(* Check controller alarm *)
IF sREL_ALM<>REL_ALM THEN
	CASE REL_ALM OF
		0: IF NOT chkREL_ST.OUT THEN LogEv(EL_Log,EO_LUXM,ID,1,''); END_IF
		1: LogEv(EL_Alarm,EO_LUXM,ID,6,'');
		2: LogEv(EL_Wrn  ,EO_LUXM,ID,4,WORD_TO_STRING(REL_A));
		3: LogEv(EL_Wrn  ,EO_LUXM,ID,5,WORD_TO_STRING(REL_A));
		4: LogEv(EL_Alarm,EO_LUXM,ID,7,WORD_TO_STRING(REL_A));
		5: LogEv(EL_Alarm,EO_LUXM,ID,8,'');
	END_CASE
	sREL_ALM:=REL_ALM;
END_IF

(* Status color *)
   IF REL_ALM=1 OR REL_ALM>3 OR chkREL_ST.OUT	THEN Status_Log:=2; Status_Vis:=COLOR_RED;
ELSIF REL_ALM<>0								THEN Status_Log:=1; Status_Vis:=COLOR_YELLOW;
                  	   							ELSE Status_Log:=0; Status_Vis:=SEL(REL_EN,COLOR_GREEN_OFF,COLOR_GREEN);
END_IF

ACTION AddLogData:
Logger.s1:=INSERT('&LUXM=',BYTE_TO_STRING(ID),5);
IF ID<10 THEN Logger.s1:=INSERT(Logger.s1,'0',5); END_IF

Logger.s1:=CONCAT(Logger.s1,WORD_TO_STRING(REL_V));				Logger.s1:=CONCAT(Logger.s1,';');
Logger.s1:=CONCAT(Logger.s1,WORD_TO_STRING(REL_A));				Logger.s1:=CONCAT(Logger.s1,';');
Logger.s1:=CONCAT(Logger.s1,DWORD_TO_STRING(ENERGYCOUNTER));	Logger.s1:=CONCAT(Logger.s1,';');
Logger.s1:=CONCAT(Logger.s1,DWORD_TO_STRING(WORKINGTIME));		Logger.s1:=CONCAT(Logger.s1,';');
Logger.s1:=CONCAT(Logger.s1,DWORD_TO_STRING(POWERONCYCLES));	Logger.s1:=CONCAT(Logger.s1,';');
Logger.s1:=CONCAT(Logger.s1,INT_TO_STRING(REL_TEMP));			Logger.s1:=CONCAT(Logger.s1,';');

Logger.s1:=CONCAT(Logger.s1,BYTE_TO_STRING(Status_Log));
ADDSTRING(ADR(Logger.TData), ADR(Logger.s1), Logger.TLen);
END_ACTION

ACTION StatReset:
(* Reset statistic counters *)
WORKINGTIME:=0;
POWERONCYCLES:=0;
ENERGYCOUNTER:=0;
END_ACTION

END_FUNCTION_BLOCK

// AC14nn/Application/VIS_CHONOEDITOR
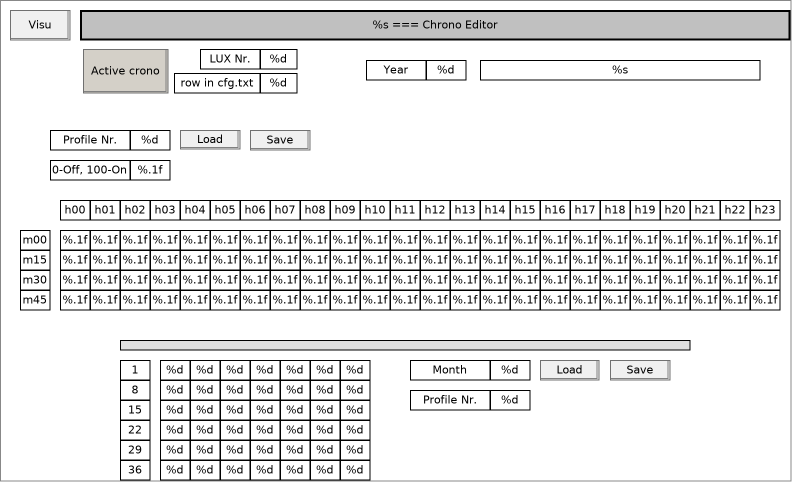
VISUALIZATION VIS_CHONOEDITOR  // 792x482
VAR_IN_OUT
//	x	: word;
//	LuxSel	: word;	
END_VAR
    Rectangle (200,49 60x20), "LUX Nr."
    Rectangle (260,49 37x20), "%d", text variable: CronEd.CN_Sel, colour toggle: CronEd.CN_Sel<>CronEd.CN_Act
        OnMouseDown: write the text variable via Edit, min 1, max 900, title '1'
    Rectangle (50,130 80x20), "Profile Nr."
    Rectangle (130,130 40x20), "%d", text variable: CronEd.PR_Sel, colour toggle: CronEd.PR_Sel<>CronEd.PR_Act
        OnMouseDown: write the text variable via Edit, min 1, max 10
    Rectangle (50,160 80x20), "0-Off, 100-On"
    Rectangle (130,160 40x20), "%.1f", text variable: CronEd.PR_TT
        OnMouseDown: write the text variable via Edit
    Button (180,130 60x19), "Load", pressed state: CronEd.PR_Load
        toggle CronEd.PR_Load
    Button (250,130 60x20), "Save", pressed state: CronEd.PR_Save
        toggle CronEd.PR_Save
    Rectangle (20,230 30x20), "m00"
    Rectangle (20,250 30x20), "m15"
    Rectangle (20,270 30x20), "m30"
    Rectangle (20,290 30x20), "m45"
    Rectangle (80,10 710x30), "%s === Chrono Editor", text variable: Plant_NAME
    Button (10,10 60x30), "Visu"
        OnMouseUp:  Assign=PLC_Visualization, Type=Assignment
    Polygon (20,210)
    RoundedRectangle (60,230 30x20), "%.1f", text variable: INT_TO_REAL(CronEd.PR.Setpoint[0])/10
        OnMouseUp: execute { CronEd.PR.Setpoint[0]:=(REAL_TO_WORD(CronEd.PR_TT*10)); }
    RoundedRectangle (60,250 30x20), "%.1f", text variable: INT_TO_REAL(CronEd.PR.Setpoint[1])/10
        OnMouseUp: execute { CronEd.PR.Setpoint[1]:=(REAL_TO_WORD(CronEd.PR_TT*10)); }
    RoundedRectangle (60,270 30x20), "%.1f", text variable: INT_TO_REAL(CronEd.PR.Setpoint[2])/10
        OnMouseUp: execute { CronEd.PR.Setpoint[2]:=(REAL_TO_WORD(CronEd.PR_TT*10)); }
    RoundedRectangle (60,290 30x20), "%.1f", text variable: INT_TO_REAL(CronEd.PR.Setpoint[3])/10
        OnMouseUp: execute { CronEd.PR.Setpoint[3]:=(REAL_TO_WORD(CronEd.PR_TT*10)); }
    Rectangle (60,200 30x20), "h00"
        OnMouseUp: execute { CronEd.PR.Setpoint[0]:=(REAL_TO_WORD(CronEd.PR_TT*10)); }
        OnMouseUp: execute { CronEd.PR.Setpoint[1]:=(REAL_TO_WORD(CronEd.PR_TT*10)); }
        OnMouseUp: execute { CronEd.PR.Setpoint[2]:=(REAL_TO_WORD(CronEd.PR_TT*10)); }
        OnMouseUp: execute { CronEd.PR.Setpoint[3]:=(REAL_TO_WORD(CronEd.PR_TT*10)); }
    RoundedRectangle (90,230 30x20), "%.1f", text variable: INT_TO_REAL(CronEd.PR.Setpoint[4])/10
        OnMouseUp: execute { CronEd.PR.Setpoint[4]:=(REAL_TO_WORD(CronEd.PR_TT*10)); }
    RoundedRectangle (90,250 30x20), "%.1f", text variable: INT_TO_REAL(CronEd.PR.Setpoint[5])/10
        OnMouseUp: execute { CronEd.PR.Setpoint[5]:=(REAL_TO_WORD(CronEd.PR_TT*10)); }
    RoundedRectangle (90,270 30x20), "%.1f", text variable: INT_TO_REAL(CronEd.PR.Setpoint[6])/10
        OnMouseUp: execute { CronEd.PR.Setpoint[6]:=(REAL_TO_WORD(CronEd.PR_TT*10)); }
    RoundedRectangle (90,290 30x20), "%.1f", text variable: INT_TO_REAL(CronEd.PR.Setpoint[7])/10
        OnMouseUp: execute { CronEd.PR.Setpoint[7]:=(REAL_TO_WORD(CronEd.PR_TT*10)); }
    Rectangle (90,200 30x20), "h01"
        OnMouseUp: execute { CronEd.PR.Setpoint[4]:=(REAL_TO_WORD(CronEd.PR_TT*10)); }
        OnMouseUp: execute { CronEd.PR.Setpoint[5]:=(REAL_TO_WORD(CronEd.PR_TT*10)); }
        OnMouseUp: execute { CronEd.PR.Setpoint[6]:=(REAL_TO_WORD(CronEd.PR_TT*10)); }
        OnMouseUp: execute { CronEd.PR.Setpoint[7]:=(REAL_TO_WORD(CronEd.PR_TT*10)); }
    RoundedRectangle (120,230 30x20), "%.1f", text variable: INT_TO_REAL(CronEd.PR.Setpoint[8])/10
        OnMouseUp: execute { CronEd.PR.Setpoint[8]:=(REAL_TO_WORD(CronEd.PR_TT*10)); }
    RoundedRectangle (120,250 30x20), "%.1f", text variable: INT_TO_REAL(CronEd.PR.Setpoint[9])/10
        OnMouseUp: execute { CronEd.PR.Setpoint[9]:=(REAL_TO_WORD(CronEd.PR_TT*10)); }
    RoundedRectangle (120,270 30x20), "%.1f", text variable: INT_TO_REAL(CronEd.PR.Setpoint[10])/10
        OnMouseUp: execute { CronEd.PR.Setpoint[10]:=(REAL_TO_WORD(CronEd.PR_TT*10)); }
    RoundedRectangle (120,290 30x20), "%.1f", text variable: INT_TO_REAL(CronEd.PR.Setpoint[11])/10
        OnMouseUp: execute { CronEd.PR.Setpoint[11]:=(REAL_TO_WORD(CronEd.PR_TT*10)); }
    Rectangle (120,200 30x20), "h02"
        OnMouseUp: execute { CronEd.PR.Setpoint[8]:=(REAL_TO_WORD(CronEd.PR_TT*10)); }
        OnMouseUp: execute { CronEd.PR.Setpoint[9]:=(REAL_TO_WORD(CronEd.PR_TT*10)); }
        OnMouseUp: execute { CronEd.PR.Setpoint[10]:=(REAL_TO_WORD(CronEd.PR_TT*10)); }
        OnMouseUp: execute { CronEd.PR.Setpoint[11]:=(REAL_TO_WORD(CronEd.PR_TT*10)); }
    RoundedRectangle (150,230 30x20), "%.1f", text variable: INT_TO_REAL(CronEd.PR.Setpoint[12])/10
        OnMouseUp: execute { CronEd.PR.Setpoint[12]:=(REAL_TO_WORD(CronEd.PR_TT*10)); }
    RoundedRectangle (150,250 30x20), "%.1f", text variable: INT_TO_REAL(CronEd.PR.Setpoint[13])/10
        OnMouseUp: execute { CronEd.PR.Setpoint[13]:=(REAL_TO_WORD(CronEd.PR_TT*10)); }
    RoundedRectangle (150,270 30x20), "%.1f", text variable: INT_TO_REAL(CronEd.PR.Setpoint[14])/10
        OnMouseUp: execute { CronEd.PR.Setpoint[14]:=(REAL_TO_WORD(CronEd.PR_TT*10)); }
    RoundedRectangle (150,290 30x20), "%.1f", text variable: INT_TO_REAL(CronEd.PR.Setpoint[15])/10
        OnMouseUp: execute { CronEd.PR.Setpoint[15]:=(REAL_TO_WORD(CronEd.PR_TT*10)); }
    Rectangle (150,200 30x20), "h03"
        OnMouseUp: execute { CronEd.PR.Setpoint[15]:=(REAL_TO_WORD(CronEd.PR_TT*10)); }
        OnMouseUp: execute { CronEd.PR.Setpoint[14]:=(REAL_TO_WORD(CronEd.PR_TT*10)); }
        OnMouseUp: execute { CronEd.PR.Setpoint[13]:=(REAL_TO_WORD(CronEd.PR_TT*10)); }
        OnMouseUp: execute { CronEd.PR.Setpoint[12]:=(REAL_TO_WORD(CronEd.PR_TT*10)); }
    RoundedRectangle (180,230 30x20), "%.1f", text variable: INT_TO_REAL(CronEd.PR.Setpoint[16])/10
        OnMouseUp: execute { CronEd.PR.Setpoint[16]:=(REAL_TO_WORD(CronEd.PR_TT*10)); }
    RoundedRectangle (180,250 30x20), "%.1f", text variable: INT_TO_REAL(CronEd.PR.Setpoint[17])/10
        OnMouseUp: execute { CronEd.PR.Setpoint[17]:=(REAL_TO_WORD(CronEd.PR_TT*10)); }
    RoundedRectangle (180,270 30x20), "%.1f", text variable: INT_TO_REAL(CronEd.PR.Setpoint[18])/10
        OnMouseUp: execute { CronEd.PR.Setpoint[18]:=(REAL_TO_WORD(CronEd.PR_TT*10)); }
    RoundedRectangle (180,290 30x20), "%.1f", text variable: INT_TO_REAL(CronEd.PR.Setpoint[19])/10
        OnMouseUp: execute { CronEd.PR.Setpoint[19]:=(REAL_TO_WORD(CronEd.PR_TT*10)); }
    Rectangle (180,200 30x20), "h04"
        OnMouseUp: execute { CronEd.PR.Setpoint[19]:=(REAL_TO_WORD(CronEd.PR_TT*10)); }
        OnMouseUp: execute { CronEd.PR.Setpoint[18]:=(REAL_TO_WORD(CronEd.PR_TT*10)); }
        OnMouseUp: execute { CronEd.PR.Setpoint[17]:=(REAL_TO_WORD(CronEd.PR_TT*10)); }
        OnMouseUp: execute { CronEd.PR.Setpoint[16]:=(REAL_TO_WORD(CronEd.PR_TT*10)); }
    RoundedRectangle (210,230 30x20), "%.1f", text variable: INT_TO_REAL(CronEd.PR.Setpoint[20])/10
        OnMouseUp: execute { CronEd.PR.Setpoint[20]:=(REAL_TO_WORD(CronEd.PR_TT*10)); }
    RoundedRectangle (210,250 30x20), "%.1f", text variable: INT_TO_REAL(CronEd.PR.Setpoint[21])/10
        OnMouseUp: execute { CronEd.PR.Setpoint[21]:=(REAL_TO_WORD(CronEd.PR_TT*10)); }
    RoundedRectangle (210,270 30x20), "%.1f", text variable: INT_TO_REAL(CronEd.PR.Setpoint[22])/10
        OnMouseUp: execute { CronEd.PR.Setpoint[22]:=(REAL_TO_WORD(CronEd.PR_TT*10)); }
    RoundedRectangle (210,290 30x20), "%.1f", text variable: INT_TO_REAL(CronEd.PR.Setpoint[23])/10
        OnMouseUp: execute { CronEd.PR.Setpoint[23]:=(REAL_TO_WORD(CronEd.PR_TT*10)); }
    Rectangle (210,200 30x20), "h05"
        OnMouseUp: execute { CronEd.PR.Setpoint[23]:=(REAL_TO_WORD(CronEd.PR_TT*10)); }
        OnMouseUp: execute { CronEd.PR.Setpoint[22]:=(REAL_TO_WORD(CronEd.PR_TT*10)); }
        OnMouseUp: execute { CronEd.PR.Setpoint[21]:=(REAL_TO_WORD(CronEd.PR_TT*10)); }
        OnMouseUp: execute { CronEd.PR.Setpoint[20]:=(REAL_TO_WORD(CronEd.PR_TT*10)); }
    RoundedRectangle (240,230 30x20), "%.1f", text variable: INT_TO_REAL(CronEd.PR.Setpoint[24])/10
        OnMouseUp: execute { CronEd.PR.Setpoint[24]:=(REAL_TO_WORD(CronEd.PR_TT*10)); }
    RoundedRectangle (240,250 30x20), "%.1f", text variable: INT_TO_REAL(CronEd.PR.Setpoint[25])/10
        OnMouseUp: execute { CronEd.PR.Setpoint[25]:=(REAL_TO_WORD(CronEd.PR_TT*10)); }
    RoundedRectangle (240,270 30x20), "%.1f", text variable: INT_TO_REAL(CronEd.PR.Setpoint[26])/10
        OnMouseUp: execute { CronEd.PR.Setpoint[26]:=(REAL_TO_WORD(CronEd.PR_TT*10)); }
    RoundedRectangle (240,290 30x20), "%.1f", text variable: INT_TO_REAL(CronEd.PR.Setpoint[27])/10
        OnMouseUp: execute { CronEd.PR.Setpoint[27]:=(REAL_TO_WORD(CronEd.PR_TT*10)); }
    Rectangle (240,200 30x20), "h06"
        OnMouseUp: execute { CronEd.PR.Setpoint[27]:=(REAL_TO_WORD(CronEd.PR_TT*10)); }
        OnMouseUp: execute { CronEd.PR.Setpoint[26]:=(REAL_TO_WORD(CronEd.PR_TT*10)); }
        OnMouseUp: execute { CronEd.PR.Setpoint[25]:=(REAL_TO_WORD(CronEd.PR_TT*10)); }
        OnMouseUp: execute { CronEd.PR.Setpoint[24]:=(REAL_TO_WORD(CronEd.PR_TT*10)); }
    RoundedRectangle (270,230 30x20), "%.1f", text variable: INT_TO_REAL(CronEd.PR.Setpoint[28])/10
        OnMouseUp: execute { CronEd.PR.Setpoint[28]:=(REAL_TO_WORD(CronEd.PR_TT*10)); }
    RoundedRectangle (270,250 30x20), "%.1f", text variable: INT_TO_REAL(CronEd.PR.Setpoint[29])/10
        OnMouseUp: execute { CronEd.PR.Setpoint[29]:=(REAL_TO_WORD(CronEd.PR_TT*10)); }
    RoundedRectangle (270,270 30x20), "%.1f", text variable: INT_TO_REAL(CronEd.PR.Setpoint[30])/10
        OnMouseUp: execute { CronEd.PR.Setpoint[30]:=(REAL_TO_WORD(CronEd.PR_TT*10)); }
    RoundedRectangle (270,290 30x20), "%.1f", text variable: INT_TO_REAL(CronEd.PR.Setpoint[31])/10
        OnMouseUp: execute { CronEd.PR.Setpoint[31]:=(REAL_TO_WORD(CronEd.PR_TT*10)); }
    Rectangle (270,200 30x20), "h07"
        OnMouseUp: execute { CronEd.PR.Setpoint[31]:=(REAL_TO_WORD(CronEd.PR_TT*10)); }
        OnMouseUp: execute { CronEd.PR.Setpoint[30]:=(REAL_TO_WORD(CronEd.PR_TT*10)); }
        OnMouseUp: execute { CronEd.PR.Setpoint[29]:=(REAL_TO_WORD(CronEd.PR_TT*10)); }
        OnMouseUp: execute { CronEd.PR.Setpoint[28]:=(REAL_TO_WORD(CronEd.PR_TT*10)); }
    RoundedRectangle (300,230 30x20), "%.1f", text variable: INT_TO_REAL(CronEd.PR.Setpoint[32])/10
        OnMouseUp: execute { CronEd.PR.Setpoint[32]:=(REAL_TO_WORD(CronEd.PR_TT*10)); }
    RoundedRectangle (300,250 30x20), "%.1f", text variable: INT_TO_REAL(CronEd.PR.Setpoint[33])/10
        OnMouseUp: execute { CronEd.PR.Setpoint[33]:=(REAL_TO_WORD(CronEd.PR_TT*10)); }
    RoundedRectangle (300,270 30x20), "%.1f", text variable: INT_TO_REAL(CronEd.PR.Setpoint[34])/10
        OnMouseUp: execute { CronEd.PR.Setpoint[34]:=(REAL_TO_WORD(CronEd.PR_TT*10)); }
    RoundedRectangle (300,290 30x20), "%.1f", text variable: INT_TO_REAL(CronEd.PR.Setpoint[35])/10
        OnMouseUp: execute { CronEd.PR.Setpoint[35]:=(REAL_TO_WORD(CronEd.PR_TT*10)); }
    Rectangle (300,200 30x20), "h08"
        OnMouseUp: execute { CronEd.PR.Setpoint[35]:=(REAL_TO_WORD(CronEd.PR_TT*10)); }
        OnMouseUp: execute { CronEd.PR.Setpoint[34]:=(REAL_TO_WORD(CronEd.PR_TT*10)); }
        OnMouseUp: execute { CronEd.PR.Setpoint[33]:=(REAL_TO_WORD(CronEd.PR_TT*10)); }
        OnMouseUp: execute { CronEd.PR.Setpoint[32]:=(REAL_TO_WORD(CronEd.PR_TT*10)); }
    RoundedRectangle (330,230 30x20), "%.1f", text variable: INT_TO_REAL(CronEd.PR.Setpoint[36])/10
        OnMouseUp: execute { CronEd.PR.Setpoint[36]:=(REAL_TO_WORD(CronEd.PR_TT*10)); }
    RoundedRectangle (330,250 30x20), "%.1f", text variable: INT_TO_REAL(CronEd.PR.Setpoint[37])/10
        OnMouseUp: execute { CronEd.PR.Setpoint[37]:=(REAL_TO_WORD(CronEd.PR_TT*10)); }
    RoundedRectangle (330,270 30x20), "%.1f", text variable: INT_TO_REAL(CronEd.PR.Setpoint[38])/10
        OnMouseUp: execute { CronEd.PR.Setpoint[38]:=(REAL_TO_WORD(CronEd.PR_TT*10)); }
    RoundedRectangle (330,290 30x20), "%.1f", text variable: INT_TO_REAL(CronEd.PR.Setpoint[39])/10
        OnMouseUp: execute { CronEd.PR.Setpoint[39]:=(REAL_TO_WORD(CronEd.PR_TT*10)); }
    Rectangle (330,200 30x20), "h09"
        OnMouseUp: execute { CronEd.PR.Setpoint[39]:=(REAL_TO_WORD(CronEd.PR_TT*10)); }
        OnMouseUp: execute { CronEd.PR.Setpoint[38]:=(REAL_TO_WORD(CronEd.PR_TT*10)); }
        OnMouseUp: execute { CronEd.PR.Setpoint[37]:=(REAL_TO_WORD(CronEd.PR_TT*10)); }
        OnMouseUp: execute { CronEd.PR.Setpoint[36]:=(REAL_TO_WORD(CronEd.PR_TT*10)); }
    RoundedRectangle (360,230 30x20), "%.1f", text variable: INT_TO_REAL(CronEd.PR.Setpoint[40])/10
        OnMouseUp: execute { CronEd.PR.Setpoint[40]:=(REAL_TO_WORD(CronEd.PR_TT*10)); }
    RoundedRectangle (360,250 30x20), "%.1f", text variable: INT_TO_REAL(CronEd.PR.Setpoint[41])/10
        OnMouseUp: execute { CronEd.PR.Setpoint[41]:=(REAL_TO_WORD(CronEd.PR_TT*10)); }
    RoundedRectangle (360,270 30x20), "%.1f", text variable: INT_TO_REAL(CronEd.PR.Setpoint[42])/10
        OnMouseUp: execute { CronEd.PR.Setpoint[42]:=(REAL_TO_WORD(CronEd.PR_TT*10)); }
    RoundedRectangle (360,290 30x20), "%.1f", text variable: INT_TO_REAL(CronEd.PR.Setpoint[43])/10
        OnMouseUp: execute { CronEd.PR.Setpoint[43]:=(REAL_TO_WORD(CronEd.PR_TT*10)); }
    Rectangle (360,200 30x20), "h10"
        OnMouseUp: execute { CronEd.PR.Setpoint[43]:=(REAL_TO_WORD(CronEd.PR_TT*10)); }
        OnMouseUp: execute { CronEd.PR.Setpoint[42]:=(REAL_TO_WORD(CronEd.PR_TT*10)); }
        OnMouseUp: execute { CronEd.PR.Setpoint[41]:=(REAL_TO_WORD(CronEd.PR_TT*10)); }
        OnMouseUp: execute { CronEd.PR.Setpoint[40]:=(REAL_TO_WORD(CronEd.PR_TT*10)); }
    RoundedRectangle (390,230 30x20), "%.1f", text variable: INT_TO_REAL(CronEd.PR.Setpoint[44])/10
        OnMouseUp: execute { CronEd.PR.Setpoint[44]:=(REAL_TO_WORD(CronEd.PR_TT*10)); }
    RoundedRectangle (390,250 30x20), "%.1f", text variable: INT_TO_REAL(CronEd.PR.Setpoint[45])/10
        OnMouseUp: execute { CronEd.PR.Setpoint[45]:=(REAL_TO_WORD(CronEd.PR_TT*10)); }
    RoundedRectangle (390,270 30x20), "%.1f", text variable: INT_TO_REAL(CronEd.PR.Setpoint[46])/10
        OnMouseUp: execute { CronEd.PR.Setpoint[46]:=(REAL_TO_WORD(CronEd.PR_TT*10)); }
    RoundedRectangle (390,290 30x20), "%.1f", text variable: INT_TO_REAL(CronEd.PR.Setpoint[47])/10
        OnMouseUp: execute { CronEd.PR.Setpoint[47]:=(REAL_TO_WORD(CronEd.PR_TT*10)); }
    Rectangle (390,200 30x20), "h11"
        OnMouseUp: execute { CronEd.PR.Setpoint[47]:=(REAL_TO_WORD(CronEd.PR_TT*10)); }
        OnMouseUp: execute { CronEd.PR.Setpoint[46]:=(REAL_TO_WORD(CronEd.PR_TT*10)); }
        OnMouseUp: execute { CronEd.PR.Setpoint[45]:=(REAL_TO_WORD(CronEd.PR_TT*10)); }
        OnMouseUp: execute { CronEd.PR.Setpoint[44]:=(REAL_TO_WORD(CronEd.PR_TT*10)); }
    RoundedRectangle (420,230 30x20), "%.1f", text variable: INT_TO_REAL(CronEd.PR.Setpoint[48])/10
        OnMouseUp: execute { CronEd.PR.Setpoint[48]:=(REAL_TO_WORD(CronEd.PR_TT*10)); }
    RoundedRectangle (420,250 30x20), "%.1f", text variable: INT_TO_REAL(CronEd.PR.Setpoint[49])/10
        OnMouseUp: execute { CronEd.PR.Setpoint[49]:=(REAL_TO_WORD(CronEd.PR_TT*10)); }
    RoundedRectangle (420,270 30x20), "%.1f", text variable: INT_TO_REAL(CronEd.PR.Setpoint[50])/10
        OnMouseUp: execute { CronEd.PR.Setpoint[50]:=(REAL_TO_WORD(CronEd.PR_TT*10)); }
    RoundedRectangle (420,290 30x20), "%.1f", text variable: INT_TO_REAL(CronEd.PR.Setpoint[51])/10
        OnMouseUp: execute { CronEd.PR.Setpoint[51]:=(REAL_TO_WORD(CronEd.PR_TT*10)); }
    Rectangle (420,200 30x20), "h12"
        OnMouseUp: execute { CronEd.PR.Setpoint[51]:=(REAL_TO_WORD(CronEd.PR_TT*10)); }
        OnMouseUp: execute { CronEd.PR.Setpoint[50]:=(REAL_TO_WORD(CronEd.PR_TT*10)); }
        OnMouseUp: execute { CronEd.PR.Setpoint[49]:=(REAL_TO_WORD(CronEd.PR_TT*10)); }
        OnMouseUp: execute { CronEd.PR.Setpoint[48]:=(REAL_TO_WORD(CronEd.PR_TT*10)); }
    RoundedRectangle (450,230 30x20), "%.1f", text variable: INT_TO_REAL(CronEd.PR.Setpoint[52])/10
        OnMouseUp: execute { CronEd.PR.Setpoint[52]:=(REAL_TO_WORD(CronEd.PR_TT*10)); }
    RoundedRectangle (450,250 30x20), "%.1f", text variable: INT_TO_REAL(CronEd.PR.Setpoint[53])/10
        OnMouseUp: execute { CronEd.PR.Setpoint[53]:=(REAL_TO_WORD(CronEd.PR_TT*10)); }
    RoundedRectangle (450,270 30x20), "%.1f", text variable: INT_TO_REAL(CronEd.PR.Setpoint[54])/10
        OnMouseUp: execute { CronEd.PR.Setpoint[54]:=(REAL_TO_WORD(CronEd.PR_TT*10)); }
    RoundedRectangle (450,290 30x20), "%.1f", text variable: INT_TO_REAL(CronEd.PR.Setpoint[55])/10
        OnMouseUp: execute { CronEd.PR.Setpoint[55]:=(REAL_TO_WORD(CronEd.PR_TT*10)); }
    Rectangle (450,200 30x20), "h13"
        OnMouseUp: execute { CronEd.PR.Setpoint[55]:=(REAL_TO_WORD(CronEd.PR_TT*10)); }
        OnMouseUp: execute { CronEd.PR.Setpoint[54]:=(REAL_TO_WORD(CronEd.PR_TT*10)); }
        OnMouseUp: execute { CronEd.PR.Setpoint[53]:=(REAL_TO_WORD(CronEd.PR_TT*10)); }
        OnMouseUp: execute { CronEd.PR.Setpoint[52]:=(REAL_TO_WORD(CronEd.PR_TT*10)); }
    RoundedRectangle (480,230 30x20), "%.1f", text variable: INT_TO_REAL(CronEd.PR.Setpoint[56])/10
        OnMouseUp: execute { CronEd.PR.Setpoint[56]:=(REAL_TO_WORD(CronEd.PR_TT*10)); }
    RoundedRectangle (480,250 30x20), "%.1f", text variable: INT_TO_REAL(CronEd.PR.Setpoint[57])/10
        OnMouseUp: execute { CronEd.PR.Setpoint[57]:=(REAL_TO_WORD(CronEd.PR_TT*10)); }
    RoundedRectangle (480,270 30x20), "%.1f", text variable: INT_TO_REAL(CronEd.PR.Setpoint[58])/10
        OnMouseUp: execute { CronEd.PR.Setpoint[58]:=(REAL_TO_WORD(CronEd.PR_TT*10)); }
    RoundedRectangle (480,290 30x20), "%.1f", text variable: INT_TO_REAL(CronEd.PR.Setpoint[59])/10
        OnMouseUp: execute { CronEd.PR.Setpoint[59]:=(REAL_TO_WORD(CronEd.PR_TT*10)); }
    Rectangle (480,200 30x20), "h14"
        OnMouseUp: execute { CronEd.PR.Setpoint[59]:=(REAL_TO_WORD(CronEd.PR_TT*10)); }
        OnMouseUp: execute { CronEd.PR.Setpoint[58]:=(REAL_TO_WORD(CronEd.PR_TT*10)); }
        OnMouseUp: execute { CronEd.PR.Setpoint[57]:=(REAL_TO_WORD(CronEd.PR_TT*10)); }
        OnMouseUp: execute { CronEd.PR.Setpoint[56]:=(REAL_TO_WORD(CronEd.PR_TT*10)); }
    RoundedRectangle (510,230 30x20), "%.1f", text variable: INT_TO_REAL(CronEd.PR.Setpoint[60])/10
        OnMouseUp: execute { CronEd.PR.Setpoint[60]:=(REAL_TO_WORD(CronEd.PR_TT*10)); }
    RoundedRectangle (510,250 30x20), "%.1f", text variable: INT_TO_REAL(CronEd.PR.Setpoint[61])/10
        OnMouseUp: execute { CronEd.PR.Setpoint[61]:=(REAL_TO_WORD(CronEd.PR_TT*10)); }
    RoundedRectangle (510,270 30x20), "%.1f", text variable: INT_TO_REAL(CronEd.PR.Setpoint[62])/10
        OnMouseUp: execute { CronEd.PR.Setpoint[62]:=(REAL_TO_WORD(CronEd.PR_TT*10)); }
    RoundedRectangle (510,290 30x20), "%.1f", text variable: INT_TO_REAL(CronEd.PR.Setpoint[63])/10
        OnMouseUp: execute { CronEd.PR.Setpoint[63]:=(REAL_TO_WORD(CronEd.PR_TT*10)); }
    Rectangle (510,200 30x20), "h15"
        OnMouseUp: execute { CronEd.PR.Setpoint[63]:=(REAL_TO_WORD(CronEd.PR_TT*10)); }
        OnMouseUp: execute { CronEd.PR.Setpoint[62]:=(REAL_TO_WORD(CronEd.PR_TT*10)); }
        OnMouseUp: execute { CronEd.PR.Setpoint[61]:=(REAL_TO_WORD(CronEd.PR_TT*10)); }
        OnMouseUp: execute { CronEd.PR.Setpoint[60]:=(REAL_TO_WORD(CronEd.PR_TT*10)); }
    RoundedRectangle (540,230 30x20), "%.1f", text variable: INT_TO_REAL(CronEd.PR.Setpoint[64])/10
        OnMouseUp: execute { CronEd.PR.Setpoint[64]:=(REAL_TO_WORD(CronEd.PR_TT*10)); }
    RoundedRectangle (540,250 30x20), "%.1f", text variable: INT_TO_REAL(CronEd.PR.Setpoint[65])/10
        OnMouseUp: execute { CronEd.PR.Setpoint[65]:=(REAL_TO_WORD(CronEd.PR_TT*10)); }
    RoundedRectangle (540,270 30x20), "%.1f", text variable: INT_TO_REAL(CronEd.PR.Setpoint[66])/10
        OnMouseUp: execute { CronEd.PR.Setpoint[66]:=(REAL_TO_WORD(CronEd.PR_TT*10)); }
    RoundedRectangle (540,290 30x20), "%.1f", text variable: INT_TO_REAL(CronEd.PR.Setpoint[67])/10
        OnMouseUp: execute { CronEd.PR.Setpoint[67]:=(REAL_TO_WORD(CronEd.PR_TT*10)); }
    Rectangle (540,200 30x20), "h16"
        OnMouseUp: execute { CronEd.PR.Setpoint[67]:=(REAL_TO_WORD(CronEd.PR_TT*10)); }
        OnMouseUp: execute { CronEd.PR.Setpoint[66]:=(REAL_TO_WORD(CronEd.PR_TT*10)); }
        OnMouseUp: execute { CronEd.PR.Setpoint[65]:=(REAL_TO_WORD(CronEd.PR_TT*10)); }
        OnMouseUp: execute { CronEd.PR.Setpoint[64]:=(REAL_TO_WORD(CronEd.PR_TT*10)); }
    RoundedRectangle (570,230 30x20), "%.1f", text variable: INT_TO_REAL(CronEd.PR.Setpoint[68])/10
        OnMouseUp: execute { CronEd.PR.Setpoint[68]:=(REAL_TO_WORD(CronEd.PR_TT*10)); }
    RoundedRectangle (570,250 30x20), "%.1f", text variable: INT_TO_REAL(CronEd.PR.Setpoint[69])/10
        OnMouseUp: execute { CronEd.PR.Setpoint[69]:=(REAL_TO_WORD(CronEd.PR_TT*10)); }
    RoundedRectangle (570,270 30x20), "%.1f", text variable: INT_TO_REAL(CronEd.PR.Setpoint[70])/10
        OnMouseUp: execute { CronEd.PR.Setpoint[70]:=(REAL_TO_WORD(CronEd.PR_TT*10)); }
    RoundedRectangle (570,290 30x20), "%.1f", text variable: INT_TO_REAL(CronEd.PR.Setpoint[71])/10
        OnMouseUp: execute { CronEd.PR.Setpoint[71]:=(REAL_TO_WORD(CronEd.PR_TT*10)); }
    Rectangle (570,200 30x20), "h17"
        OnMouseUp: execute { CronEd.PR.Setpoint[71]:=(REAL_TO_WORD(CronEd.PR_TT*10)); }
        OnMouseUp: execute { CronEd.PR.Setpoint[70]:=(REAL_TO_WORD(CronEd.PR_TT*10)); }
        OnMouseUp: execute { CronEd.PR.Setpoint[69]:=(REAL_TO_WORD(CronEd.PR_TT*10)); }
        OnMouseUp: execute { CronEd.PR.Setpoint[68]:=(REAL_TO_WORD(CronEd.PR_TT*10)); }
    RoundedRectangle (600,230 30x20), "%.1f", text variable: INT_TO_REAL(CronEd.PR.Setpoint[72])/10
        OnMouseUp: execute { CronEd.PR.Setpoint[72]:=(REAL_TO_WORD(CronEd.PR_TT*10)); }
    RoundedRectangle (600,250 30x20), "%.1f", text variable: INT_TO_REAL(CronEd.PR.Setpoint[73])/10
        OnMouseUp: execute { CronEd.PR.Setpoint[73]:=(REAL_TO_WORD(CronEd.PR_TT*10)); }
    RoundedRectangle (600,270 30x20), "%.1f", text variable: INT_TO_REAL(CronEd.PR.Setpoint[74])/10
        OnMouseUp: execute { CronEd.PR.Setpoint[74]:=(REAL_TO_WORD(CronEd.PR_TT*10)); }
    RoundedRectangle (600,290 30x20), "%.1f", text variable: INT_TO_REAL(CronEd.PR.Setpoint[75])/10
        OnMouseUp: execute { CronEd.PR.Setpoint[75]:=(REAL_TO_WORD(CronEd.PR_TT*10)); }
    Rectangle (600,200 30x20), "h18"
        OnMouseUp: execute { CronEd.PR.Setpoint[75]:=(REAL_TO_WORD(CronEd.PR_TT*10)); }
        OnMouseUp: execute { CronEd.PR.Setpoint[74]:=(REAL_TO_WORD(CronEd.PR_TT*10)); }
        OnMouseUp: execute { CronEd.PR.Setpoint[73]:=(REAL_TO_WORD(CronEd.PR_TT*10)); }
        OnMouseUp: execute { CronEd.PR.Setpoint[72]:=(REAL_TO_WORD(CronEd.PR_TT*10)); }
    RoundedRectangle (630,230 30x20), "%.1f", text variable: INT_TO_REAL(CronEd.PR.Setpoint[76])/10
        OnMouseUp: execute { CronEd.PR.Setpoint[76]:=(REAL_TO_WORD(CronEd.PR_TT*10)); }
    RoundedRectangle (630,250 30x20), "%.1f", text variable: INT_TO_REAL(CronEd.PR.Setpoint[77])/10
        OnMouseUp: execute { CronEd.PR.Setpoint[77]:=(REAL_TO_WORD(CronEd.PR_TT*10)); }
    RoundedRectangle (630,270 30x20), "%.1f", text variable: INT_TO_REAL(CronEd.PR.Setpoint[78])/10
        OnMouseUp: execute { CronEd.PR.Setpoint[78]:=(REAL_TO_WORD(CronEd.PR_TT*10)); }
    RoundedRectangle (630,290 30x20), "%.1f", text variable: INT_TO_REAL(CronEd.PR.Setpoint[79])/10
        OnMouseUp: execute { CronEd.PR.Setpoint[79]:=(REAL_TO_WORD(CronEd.PR_TT*10)); }
    Rectangle (630,200 30x20), "h19"
        OnMouseUp: execute { CronEd.PR.Setpoint[79]:=(REAL_TO_WORD(CronEd.PR_TT*10)); }
        OnMouseUp: execute { CronEd.PR.Setpoint[78]:=(REAL_TO_WORD(CronEd.PR_TT*10)); }
        OnMouseUp: execute { CronEd.PR.Setpoint[77]:=(REAL_TO_WORD(CronEd.PR_TT*10)); }
        OnMouseUp: execute { CronEd.PR.Setpoint[76]:=(REAL_TO_WORD(CronEd.PR_TT*10)); }
    RoundedRectangle (660,230 30x20), "%.1f", text variable: INT_TO_REAL(CronEd.PR.Setpoint[80])/10
        OnMouseUp: execute { CronEd.PR.Setpoint[80]:=(REAL_TO_WORD(CronEd.PR_TT*10)); }
    RoundedRectangle (660,250 30x20), "%.1f", text variable: INT_TO_REAL(CronEd.PR.Setpoint[81])/10
        OnMouseUp: execute { CronEd.PR.Setpoint[81]:=(REAL_TO_WORD(CronEd.PR_TT*10)); }
    RoundedRectangle (660,270 30x20), "%.1f", text variable: INT_TO_REAL(CronEd.PR.Setpoint[82])/10
        OnMouseUp: execute { CronEd.PR.Setpoint[82]:=(REAL_TO_WORD(CronEd.PR_TT*10)); }
    RoundedRectangle (660,290 30x20), "%.1f", text variable: INT_TO_REAL(CronEd.PR.Setpoint[83])/10
        OnMouseUp: execute { CronEd.PR.Setpoint[83]:=(REAL_TO_WORD(CronEd.PR_TT*10)); }
    Rectangle (660,200 30x20), "h20"
        OnMouseUp: execute { CronEd.PR.Setpoint[83]:=(REAL_TO_WORD(CronEd.PR_TT*10)); }
        OnMouseUp: execute { CronEd.PR.Setpoint[82]:=(REAL_TO_WORD(CronEd.PR_TT*10)); }
        OnMouseUp: execute { CronEd.PR.Setpoint[81]:=(REAL_TO_WORD(CronEd.PR_TT*10)); }
        OnMouseUp: execute { CronEd.PR.Setpoint[80]:=(REAL_TO_WORD(CronEd.PR_TT*10)); }
    RoundedRectangle (690,230 30x20), "%.1f", text variable: INT_TO_REAL(CronEd.PR.Setpoint[84])/10
        OnMouseUp: execute { CronEd.PR.Setpoint[84]:=(REAL_TO_WORD(CronEd.PR_TT*10)); }
    RoundedRectangle (690,250 30x20), "%.1f", text variable: INT_TO_REAL(CronEd.PR.Setpoint[85])/10
        OnMouseUp: execute { CronEd.PR.Setpoint[85]:=(REAL_TO_WORD(CronEd.PR_TT*10)); }
    RoundedRectangle (690,270 30x20), "%.1f", text variable: INT_TO_REAL(CronEd.PR.Setpoint[86])/10
        OnMouseUp: execute { CronEd.PR.Setpoint[86]:=(REAL_TO_WORD(CronEd.PR_TT*10)); }
    RoundedRectangle (690,290 30x20), "%.1f", text variable: INT_TO_REAL(CronEd.PR.Setpoint[87])/10
        OnMouseUp: execute { CronEd.PR.Setpoint[87]:=(REAL_TO_WORD(CronEd.PR_TT*10)); }
    Rectangle (690,200 30x20), "h21"
        OnMouseUp: execute { CronEd.PR.Setpoint[87]:=(REAL_TO_WORD(CronEd.PR_TT*10)); }
        OnMouseUp: execute { CronEd.PR.Setpoint[86]:=(REAL_TO_WORD(CronEd.PR_TT*10)); }
        OnMouseUp: execute { CronEd.PR.Setpoint[85]:=(REAL_TO_WORD(CronEd.PR_TT*10)); }
        OnMouseUp: execute { CronEd.PR.Setpoint[84]:=(REAL_TO_WORD(CronEd.PR_TT*10)); }
    RoundedRectangle (720,230 30x20), "%.1f", text variable: INT_TO_REAL(CronEd.PR.Setpoint[88])/10
        OnMouseUp: execute { CronEd.PR.Setpoint[88]:=(REAL_TO_WORD(CronEd.PR_TT*10)); }
    RoundedRectangle (720,250 30x20), "%.1f", text variable: INT_TO_REAL(CronEd.PR.Setpoint[89])/10
        OnMouseUp: execute { CronEd.PR.Setpoint[89]:=(REAL_TO_WORD(CronEd.PR_TT*10)); }
    RoundedRectangle (720,270 30x20), "%.1f", text variable: INT_TO_REAL(CronEd.PR.Setpoint[90])/10
        OnMouseUp: execute { CronEd.PR.Setpoint[90]:=(REAL_TO_WORD(CronEd.PR_TT*10)); }
    RoundedRectangle (720,290 30x20), "%.1f", text variable: INT_TO_REAL(CronEd.PR.Setpoint[91])/10
        OnMouseUp: execute { CronEd.PR.Setpoint[91]:=(REAL_TO_WORD(CronEd.PR_TT*10)); }
    Rectangle (720,200 30x20), "h22"
        OnMouseUp: execute { CronEd.PR.Setpoint[91]:=(REAL_TO_WORD(CronEd.PR_TT*10)); }
        OnMouseUp: execute { CronEd.PR.Setpoint[90]:=(REAL_TO_WORD(CronEd.PR_TT*10)); }
        OnMouseUp: execute { CronEd.PR.Setpoint[89]:=(REAL_TO_WORD(CronEd.PR_TT*10)); }
        OnMouseUp: execute { CronEd.PR.Setpoint[88]:=(REAL_TO_WORD(CronEd.PR_TT*10)); }
    RoundedRectangle (750,230 30x20), "%.1f", text variable: INT_TO_REAL(CronEd.PR.Setpoint[92])/10
        OnMouseUp: execute { CronEd.PR.Setpoint[92]:=(REAL_TO_WORD(CronEd.PR_TT*10)); }
    RoundedRectangle (750,250 30x20), "%.1f", text variable: INT_TO_REAL(CronEd.PR.Setpoint[93])/10
        OnMouseUp: execute { CronEd.PR.Setpoint[93]:=(REAL_TO_WORD(CronEd.PR_TT*10)); }
    RoundedRectangle (750,270 30x20), "%.1f", text variable: INT_TO_REAL(CronEd.PR.Setpoint[94])/10
        OnMouseUp: execute { CronEd.PR.Setpoint[94]:=(REAL_TO_WORD(CronEd.PR_TT*10)); }
    RoundedRectangle (750,290 30x20), "%.1f", text variable: INT_TO_REAL(CronEd.PR.Setpoint[95])/10
        OnMouseUp: execute { CronEd.PR.Setpoint[95]:=(REAL_TO_WORD(CronEd.PR_TT*10)); }
    Rectangle (750,200 30x20), "h23"
        OnMouseUp: execute { CronEd.PR.Setpoint[95]:=(REAL_TO_WORD(CronEd.PR_TT*10)); }
        OnMouseUp: execute { CronEd.PR.Setpoint[94]:=(REAL_TO_WORD(CronEd.PR_TT*10)); }
        OnMouseUp: execute { CronEd.PR.Setpoint[93]:=(REAL_TO_WORD(CronEd.PR_TT*10)); }
        OnMouseUp: execute { CronEd.PR.Setpoint[92]:=(REAL_TO_WORD(CronEd.PR_TT*10)); }
    Rectangle (410,360 80x20), "Month"
    Rectangle (490,360 40x20), "%d", text variable: CronEd.CA_Sel, colour toggle: CronEd.CA_Sel<>CronEd.CA_Act
        OnMouseDown: write the text variable via Edit, min 1, max 12
    Rectangle (410,390 80x20), "Profile Nr."
    Rectangle (490,390 40x20), "%d", text variable: CronEd.CA_TPR
        OnMouseDown: write the text variable via Edit, min 0, max 10
    Button (540,360 59x20), "Load", pressed state: CronEd.CA_Load
        toggle CronEd.CA_Load
    Button (610,360 60x20), "Save", pressed state: CronEd.CA_Save
        toggle CronEd.CA_Save
    RoundedRectangle (160,360 30x20), "%d", text variable: CronEd.CA.Profile[0], colour toggle: CronEd.CA.Profile[0]=0, invisible if: CronEd.CA_DayF>0
        OnMouseUp: execute { CronEd.CA.Profile[0]:=(CronEd.CA_TPR); }
    Rectangle (120,360 30x20), "1"
    RoundedRectangle (190,360 30x20), "%d", text variable: CronEd.CA.Profile[1], colour toggle: CronEd.CA.Profile[1]=0, invisible if: CronEd.CA_DayF>1
        OnMouseUp: execute { CronEd.CA.Profile[1]:=(CronEd.CA_TPR); }
    RoundedRectangle (220,360 30x20), "%d", text variable: CronEd.CA.Profile[2], colour toggle: CronEd.CA.Profile[2]=0, invisible if: CronEd.CA_DayF>2
        OnMouseUp: execute { CronEd.CA.Profile[2]:=(CronEd.CA_TPR); }
    RoundedRectangle (250,360 30x20), "%d", text variable: CronEd.CA.Profile[3], colour toggle: CronEd.CA.Profile[3]=0, invisible if: CronEd.CA_DayF>3
        OnMouseUp: execute { CronEd.CA.Profile[3]:=(CronEd.CA_TPR); }
    RoundedRectangle (280,360 30x20), "%d", text variable: CronEd.CA.Profile[4], colour toggle: CronEd.CA.Profile[4]=0, invisible if: CronEd.CA_DayF>4
        OnMouseUp: execute { CronEd.CA.Profile[4]:=(CronEd.CA_TPR); }
    RoundedRectangle (310,360 30x20), "%d", text variable: CronEd.CA.Profile[5], colour toggle: CronEd.CA.Profile[5]=0, invisible if: CronEd.CA_DayF>5
        OnMouseUp: execute { CronEd.CA.Profile[5]:=(CronEd.CA_TPR); }
    RoundedRectangle (340,360 30x20), "%d", text variable: CronEd.CA.Profile[6], colour toggle: CronEd.CA.Profile[6]=0
        OnMouseUp: execute { CronEd.CA.Profile[6]:=(CronEd.CA_TPR); }
    RoundedRectangle (160,380 30x20), "%d", text variable: CronEd.CA.Profile[7], colour toggle: CronEd.CA.Profile[7]=0
        OnMouseUp: execute { CronEd.CA.Profile[7]:=(CronEd.CA_TPR); }
    Rectangle (120,380 30x20), "8"
    RoundedRectangle (190,380 30x20), "%d", text variable: CronEd.CA.Profile[8], colour toggle: CronEd.CA.Profile[8]=0
        OnMouseUp: execute { CronEd.CA.Profile[8]:=(CronEd.CA_TPR); }
    RoundedRectangle (220,380 30x20), "%d", text variable: CronEd.CA.Profile[9], colour toggle: CronEd.CA.Profile[9]=0
        OnMouseUp: execute { CronEd.CA.Profile[9]:=(CronEd.CA_TPR); }
    RoundedRectangle (250,380 30x20), "%d", text variable: CronEd.CA.Profile[10], colour toggle: CronEd.CA.Profile[10]=0
        OnMouseUp: execute { CronEd.CA.Profile[10]:=(CronEd.CA_TPR); }
    RoundedRectangle (280,380 30x20), "%d", text variable: CronEd.CA.Profile[11], colour toggle: CronEd.CA.Profile[11]=0
        OnMouseUp: execute { CronEd.CA.Profile[11]:=(CronEd.CA_TPR); }
    RoundedRectangle (310,380 30x20), "%d", text variable: CronEd.CA.Profile[12], colour toggle: CronEd.CA.Profile[12]=0
        OnMouseUp: execute { CronEd.CA.Profile[12]:=(CronEd.CA_TPR); }
    RoundedRectangle (340,380 30x20), "%d", text variable: CronEd.CA.Profile[13], colour toggle: CronEd.CA.Profile[13]=0
        OnMouseUp: execute { CronEd.CA.Profile[13]:=(CronEd.CA_TPR); }
    RoundedRectangle (160,400 30x20), "%d", text variable: CronEd.CA.Profile[14], colour toggle: CronEd.CA.Profile[14]=0
        OnMouseUp: execute { CronEd.CA.Profile[14]:=(CronEd.CA_TPR); }
    Rectangle (120,400 30x20), "15"
    RoundedRectangle (190,400 30x20), "%d", text variable: CronEd.CA.Profile[15], colour toggle: CronEd.CA.Profile[15]=0
        OnMouseUp: execute { CronEd.CA.Profile[15]:=(CronEd.CA_TPR); }
    RoundedRectangle (220,400 30x20), "%d", text variable: CronEd.CA.Profile[16], colour toggle: CronEd.CA.Profile[16]=0
        OnMouseUp: execute { CronEd.CA.Profile[16]:=(CronEd.CA_TPR); }
    RoundedRectangle (250,400 30x20), "%d", text variable: CronEd.CA.Profile[17], colour toggle: CronEd.CA.Profile[17]=0
        OnMouseUp: execute { CronEd.CA.Profile[17]:=(CronEd.CA_TPR); }
    RoundedRectangle (280,400 30x20), "%d", text variable: CronEd.CA.Profile[18], colour toggle: CronEd.CA.Profile[18]=0
        OnMouseUp: execute { CronEd.CA.Profile[18]:=(CronEd.CA_TPR); }
    RoundedRectangle (310,400 30x20), "%d", text variable: CronEd.CA.Profile[19], colour toggle: CronEd.CA.Profile[19]=0
        OnMouseUp: execute { CronEd.CA.Profile[19]:=(CronEd.CA_TPR); }
    RoundedRectangle (340,400 30x20), "%d", text variable: CronEd.CA.Profile[20], colour toggle: CronEd.CA.Profile[20]=0
        OnMouseUp: execute { CronEd.CA.Profile[20]:=(CronEd.CA_TPR); }
    RoundedRectangle (160,420 30x20), "%d", text variable: CronEd.CA.Profile[21], colour toggle: CronEd.CA.Profile[21]=0
        OnMouseUp: execute { CronEd.CA.Profile[21]:=(CronEd.CA_TPR); }
    Rectangle (120,420 30x20), "22"
    RoundedRectangle (190,420 30x20), "%d", text variable: CronEd.CA.Profile[22], colour toggle: CronEd.CA.Profile[22]=0
        OnMouseUp: execute { CronEd.CA.Profile[22]:=(CronEd.CA_TPR); }
    RoundedRectangle (220,420 30x20), "%d", text variable: CronEd.CA.Profile[23], colour toggle: CronEd.CA.Profile[23]=0
        OnMouseUp: execute { CronEd.CA.Profile[23]:=(CronEd.CA_TPR); }
    RoundedRectangle (250,420 30x20), "%d", text variable: CronEd.CA.Profile[24], colour toggle: CronEd.CA.Profile[24]=0
        OnMouseUp: execute { CronEd.CA.Profile[24]:=(CronEd.CA_TPR); }
    RoundedRectangle (280,420 30x20), "%d", text variable: CronEd.CA.Profile[25], colour toggle: CronEd.CA.Profile[25]=0
        OnMouseUp: execute { CronEd.CA.Profile[25]:=(CronEd.CA_TPR); }
    RoundedRectangle (310,420 30x20), "%d", text variable: CronEd.CA.Profile[26], colour toggle: CronEd.CA.Profile[26]=0
        OnMouseUp: execute { CronEd.CA.Profile[26]:=(CronEd.CA_TPR); }
    RoundedRectangle (340,420 30x20), "%d", text variable: CronEd.CA.Profile[27], colour toggle: CronEd.CA.Profile[27]=0
        OnMouseUp: execute { CronEd.CA.Profile[27]:=(CronEd.CA_TPR); }
    RoundedRectangle (160,440 30x20), "%d", text variable: CronEd.CA.Profile[28], colour toggle: CronEd.CA.Profile[28]=0
        OnMouseUp: execute { CronEd.CA.Profile[28]:=(CronEd.CA_TPR); }
    Rectangle (120,440 30x20), "29"
    RoundedRectangle (190,440 30x20), "%d", text variable: CronEd.CA.Profile[29], colour toggle: CronEd.CA.Profile[29]=0
        OnMouseUp: execute { CronEd.CA.Profile[29]:=(CronEd.CA_TPR); }
    RoundedRectangle (220,440 30x20), "%d", text variable: CronEd.CA.Profile[30], colour toggle: CronEd.CA.Profile[30]=0
        OnMouseUp: execute { CronEd.CA.Profile[30]:=(CronEd.CA_TPR); }
    RoundedRectangle (250,440 30x20), "%d", text variable: CronEd.CA.Profile[31], colour toggle: CronEd.CA.Profile[31]=0
        OnMouseUp: execute { CronEd.CA.Profile[31]:=(CronEd.CA_TPR); }
    RoundedRectangle (280,440 30x20), "%d", text variable: CronEd.CA.Profile[32], colour toggle: CronEd.CA.Profile[32]=0, invisible if: CronEd.CA_DayL<32
        OnMouseUp: execute { CronEd.CA.Profile[32]:=(CronEd.CA_TPR); }
    RoundedRectangle (310,440 30x20), "%d", text variable: CronEd.CA.Profile[33], colour toggle: CronEd.CA.Profile[33]=0, invisible if: CronEd.CA_DayL<33
        OnMouseUp: execute { CronEd.CA.Profile[33]:=(CronEd.CA_TPR); }
    RoundedRectangle (340,440 30x20), "%d", text variable: CronEd.CA.Profile[34], colour toggle: CronEd.CA.Profile[34]=0, invisible if: CronEd.CA_DayL<34
        OnMouseUp: execute { CronEd.CA.Profile[34]:=(CronEd.CA_TPR); }
    RoundedRectangle (160,460 30x20), "%d", text variable: CronEd.CA.Profile[35], colour toggle: CronEd.CA.Profile[35]=0, invisible if: CronEd.CA_DayL<35
        OnMouseUp: execute { CronEd.CA.Profile[35]:=(CronEd.CA_TPR); }
    Rectangle (120,460 30x20), "36", invisible if: CronEd.CA_DayL<35
    RoundedRectangle (190,460 30x20), "%d", text variable: CronEd.CA.Profile[36], colour toggle: CronEd.CA.Profile[36]=0, invisible if: CronEd.CA_DayL<36
        OnMouseUp: execute { CronEd.CA.Profile[36]:=(CronEd.CA_TPR); }
    RoundedRectangle (220,460 30x20), "%d", text variable: CronEd.CA.Profile[37], colour toggle: CronEd.CA.Profile[37]=0, invisible if: CronEd.CA_DayL<37
        OnMouseUp: execute { CronEd.CA.Profile[37]:=(CronEd.CA_TPR); }
    RoundedRectangle (250,460 30x20), "%d", text variable: CronEd.CA.Profile[38], colour toggle: CronEd.CA.Profile[38]=0, invisible if: CronEd.CA_DayL<38
        OnMouseUp: execute { CronEd.CA.Profile[38]:=(CronEd.CA_TPR); }
    RoundedRectangle (280,460 30x20), "%d", text variable: CronEd.CA.Profile[39], colour toggle: CronEd.CA.Profile[39]=0, invisible if: CronEd.CA_DayL<39
        OnMouseUp: execute { CronEd.CA.Profile[39]:=(CronEd.CA_TPR); }
    RoundedRectangle (310,460 30x20), "%d", text variable: CronEd.CA.Profile[40], colour toggle: CronEd.CA.Profile[40]=0, invisible if: CronEd.CA_DayL<40
        OnMouseUp: execute { CronEd.CA.Profile[40]:=(CronEd.CA_TPR); }
    RoundedRectangle (340,460 30x20), "%d", text variable: CronEd.CA.Profile[41], colour toggle: CronEd.CA.Profile[41]=0, invisible if: CronEd.CA_DayL<41
        OnMouseUp: execute { CronEd.CA.Profile[41]:=(CronEd.CA_TPR); }
    Rectangle (366,60 60x20), "Year"
    Rectangle (426,60 40x20), "%d", text variable: CronEd.CN_YSel, colour toggle: CronEd.CN_YSel<>CronEd.CN_YAct
        OnMouseDown: write the text variable via Edit, min 2000, max 2100, title '1'
    Rectangle (120,340 570x10)
    Rectangle (480,60 280x20), "%s", text variable: CronEd.Message
    Button (83,49 85x44), "Active crono"
        OnMouseClick: execute {
            CRON[CronEd.CN_Act].InitOK:=FALSE;
            (*	for x:= 1 to CRON_MAX do
            		if LuxElement[x].ID = CronEd.CN_Sel then
            			CronEd.CN_Act:=x;
            			CRON[CronEd.CN_Act].InitOK:=FALSE;
            			x:= CRON_MAX;
            		end_if
            	end_for
            *)
        }
    Rectangle (260,73 37x20), "%d", text variable: CronEd.CN_Act, colour toggle: CronEd.CN_Sel<>CronEd.CN_Act, invisible if: CronEd.Invisible
    Rectangle (174,73 86x20), "row in cfg.txt"
END_VISUALIZATION

// AC14nn/Application/PLC_FileManager
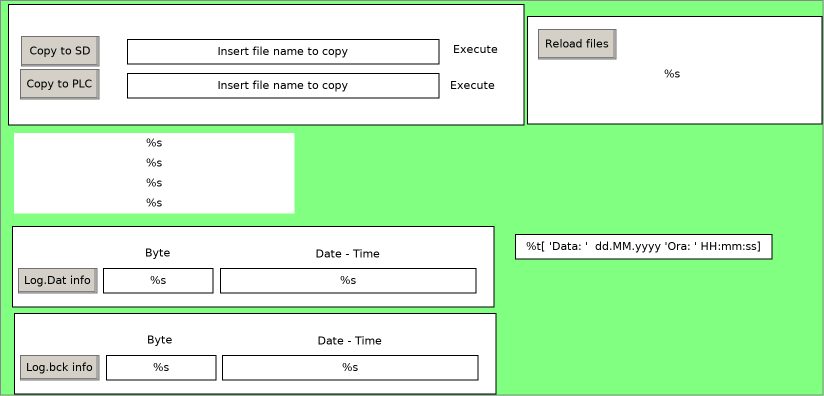
VISUALIZATION PLC_FileManager  // 824x396
    RoundedRectangle (12,226 482x81)
    RoundedRectangle (527,16 295x108)
    RoundedRectangle (8,4 516x121)
    Button (21,36 78x30), "Copy to SD"
        OnMouseClick:  ToggleVariable=PLC_PRG.CopyToSd
    Rectangle (127,39 312x25), "Insert file name to copy", text variable: PLC_PRG.FileCopyToSD.SourceFile
        OnMouseClick:  ToggleVariable=PLC_PRG.FileCopyToSD.FileCopying
        OnMouseUp: write the text variable via Edit
    Label (447,39 57x21), "Execute", invisible if: not(PLC_PRG.FileCopyToSD.FileCopying)
    Rectangle (127,73 312x25), "Insert file name to copy", text variable: PLC_PRG.FileCopySDToPLC.SourceFile
        OnMouseClick:  ToggleVariable=PLC_PRG.FileCopySDToPLC.FileCopying
        OnMouseUp: write the text variable via Edit
    Button (20,69 79x30), "Copy to PLC"
        OnMouseClick:  ToggleVariable=PLC_PRG.CopyToPLC
    Label (444,75 57x21), "Execute", invisible if: not(PLC_PRG.FileCopySDToPLC.FileCopying)
    Rectangle (14,133 280x20), "%s", text variable: PLC_PRG.OpenFileASI_PSG.Message
    Rectangle (14,153 280x20), "%s", text variable: PLC_PRG.OpenFileASI_LUX.Message
    Rectangle (14,173 280x20), "%s", text variable: PLC_PRG.OpenFileLUX_PSG.Message
    Rectangle (14,193 280x20), "%s", text variable: PLC_PRG.OpenFiles_Default_LUX.Message
    Button (538,29 78x30), "Reload files"
        OnMouseClick:  ToggleVariable=PLC_PRG.ReLoadFiles
    Rectangle (538,64 268x20), "%s", text variable: PLC_PRG.Message
    Button (18,268 79x25), "Log.Dat info"
        OnMouseClick:  ToggleVariable=PLC_PRG.FileTime
    Rectangle (220,268 256x25), "%s", text variable: PLC_PRG.FileSize_and_Time.LastModifyS
    Rectangle (103,268 110x25), "%s", text variable: PLC_PRG.FileSize_and_Time.Message
    Rectangle (103,243 110x20), "Byte"
    Rectangle (220,244 256x20), "Date - Time"
    Rectangle (515,234 257x25), "%t[ 'Data: ' dd.MM.yyyy 'Ora: ' HH:mm:ss]"
    RoundedRectangle (14,313 482x81)
    Button (20,355 79x25), "Log.bck info"
        OnMouseClick:  ToggleVariable=PLC_PRG.FileTime
    Rectangle (222,355 256x25), "%s", text variable: PLC_PRG.FileSize_and_Time.LastModifySBK
    Rectangle (105,330 110x20), "Byte"
    Rectangle (222,331 256x20), "Date - Time"
    Rectangle (106,355 110x25), "%s", text variable: PLC_PRG.FileSize_and_Time.MessageBK
END_VISUALIZATION

// AC14nn/Application/PLC_Visualization
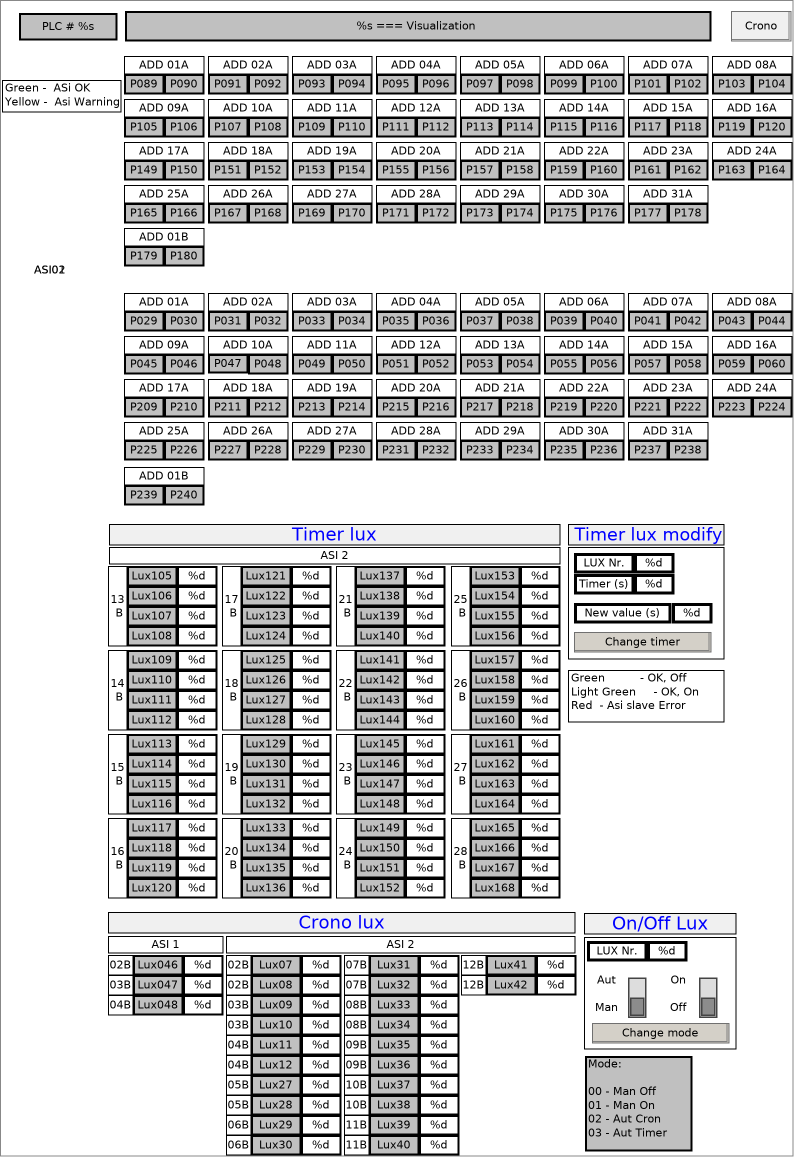
VISUALIZATION PLC_Visualization  // 794x1157
    Polygon (50,270), "ASI01", colour variable: ASI01.Status_Vis
    Polygon (50,270), "ASI02", colour variable: ASI02.Status_Vis
    Rectangle (124,311 40x20), "P029", colour variable: DataPsgForVis[29].VisStatus
    Rectangle (164,311 40x20), "P030", colour variable: DataPsgForVis[30].VisStatus
    Rectangle (124,293 80x18), "ADD 01A", colour toggle: ASI02.Asi_DeviceA[1]
    Rectangle (208,311 40x20), "P031", colour variable: DataPsgForVis[31].VisStatus
    Rectangle (248,311 40x20), "P032", colour variable: DataPsgForVis[32].VisStatus
    Rectangle (208,293 80x18), "ADD 02A", colour toggle: ASI02.Asi_DeviceA[2]
    Rectangle (292,311 40x20), "P033", colour variable: DataPsgForVis[33].VisStatus
    Rectangle (332,311 40x20), "P034", colour variable: DataPsgForVis[34].VisStatus
    Rectangle (292,293 80x18), "ADD 03A", colour toggle: ASI02.Asi_DeviceA[3]
    Rectangle (376,311 40x20), "P035", colour variable: DataPsgForVis[35].VisStatus
    Rectangle (416,311 40x20), "P036", colour variable: DataPsgForVis[36].VisStatus
    Rectangle (376,293 80x18), "ADD 04A", colour toggle: ASI02.Asi_DeviceA[4]
    Rectangle (460,311 40x20), "P037", colour variable: DataPsgForVis[37].VisStatus
    Rectangle (500,311 40x20), "P038", colour variable: DataPsgForVis[38].VisStatus
    Rectangle (460,293 80x18), "ADD 05A", colour toggle: ASI02.Asi_DeviceA[5]
    Rectangle (544,311 40x20), "P039", colour variable: DataPsgForVis[39].VisStatus
    Rectangle (584,311 40x20), "P040", colour variable: DataPsgForVis[40].VisStatus
    Rectangle (544,293 80x18), "ADD 06A", colour toggle: ASI02.Asi_DeviceA[6]
    Rectangle (628,311 40x20), "P041", colour variable: DataPsgForVis[41].VisStatus
    Rectangle (668,311 40x20), "P042", colour variable: DataPsgForVis[42].VisStatus
    Rectangle (628,293 80x18), "ADD 07A", colour toggle: ASI02.Asi_DeviceA[7]
    Rectangle (712,311 40x20), "P043", colour variable: DataPsgForVis[43].VisStatus
    Rectangle (752,311 40x20), "P044", colour variable: DataPsgForVis[44].VisStatus
    Rectangle (712,293 80x18), "ADD 08A", colour toggle: ASI02.Asi_DeviceA[8]
    Rectangle (124,354 40x20), "P045", colour variable: DataPsgForVis[45].VisStatus
    Rectangle (164,354 40x20), "P046", colour variable: DataPsgForVis[46].VisStatus
    Rectangle (124,336 80x18), "ADD 09A", colour toggle: ASI02.Asi_DeviceA[9]
    Rectangle (208,354 40x19), "P047", colour variable: DataPsgForVis[47].VisStatus
    Rectangle (248,354 40x20), "P048", colour variable: DataPsgForVis[48].VisStatus
    Rectangle (208,336 80x18), "ADD 10A", colour toggle: ASI02.Asi_DeviceA[10]
    Rectangle (292,354 40x20), "P049", colour variable: DataPsgForVis[49].VisStatus
    Rectangle (332,354 40x20), "P050", colour variable: DataPsgForVis[50].VisStatus
    Rectangle (292,336 80x18), "ADD 11A", colour toggle: ASI02.Asi_DeviceA[11]
    Rectangle (376,354 40x20), "P051", colour variable: DataPsgForVis[51].VisStatus
    Rectangle (416,354 40x20), "P052", colour variable: DataPsgForVis[52].VisStatus
    Rectangle (376,336 80x18), "ADD 12A", colour toggle: ASI02.Asi_DeviceA[12]
    Rectangle (460,354 40x20), "P053", colour variable: DataPsgForVis[53].VisStatus
    Rectangle (500,354 40x20), "P054", colour variable: DataPsgForVis[54].VisStatus
    Rectangle (460,336 80x18), "ADD 13A", colour toggle: ASI02.Asi_DeviceA[13]
    Rectangle (544,354 40x20), "P055", colour variable: DataPsgForVis[55].VisStatus
    Rectangle (584,354 40x20), "P056", colour variable: DataPsgForVis[56].VisStatus
    Rectangle (544,336 80x18), "ADD 14A", colour toggle: ASI02.Asi_DeviceA[14]
    Rectangle (628,354 40x20), "P057", colour variable: DataPsgForVis[57].VisStatus
    Rectangle (668,354 40x20), "P058", colour variable: DataPsgForVis[58].VisStatus
    Rectangle (628,336 80x18), "ADD 15A", colour toggle: ASI02.Asi_DeviceA[15]
    Rectangle (712,354 40x20), "P059", colour variable: DataPsgForVis[59].VisStatus
    Rectangle (752,354 40x20), "P060", colour variable: DataPsgForVis[60].VisStatus
    Rectangle (712,336 80x18), "ADD 16A", colour toggle: ASI02.Asi_DeviceA[16]
    Rectangle (124,397 40x20), "P209", colour variable: DataPsgForVis[209].VisStatus
    Rectangle (164,397 40x20), "P210", colour variable: DataPsgForVis[210].VisStatus
    Rectangle (124,379 80x18), "ADD 17A", colour toggle: ASI02.Asi_DeviceA[17]
    Rectangle (208,397 40x20), "P211", colour variable: DataPsgForVis[211].VisStatus
    Rectangle (248,397 40x20), "P212", colour variable: DataPsgForVis[212].VisStatus
    Rectangle (208,379 80x18), "ADD 18A", colour toggle: ASI02.Asi_DeviceA[18]
    Rectangle (292,397 40x20), "P213", colour variable: DataPsgForVis[213].VisStatus
    Rectangle (332,397 40x20), "P214", colour variable: DataPsgForVis[214].VisStatus
    Rectangle (292,379 80x18), "ADD 19A", colour toggle: ASI02.Asi_DeviceA[19]
    Rectangle (376,397 40x20), "P215", colour variable: DataPsgForVis[215].VisStatus
    Rectangle (416,397 40x20), "P216", colour variable: DataPsgForVis[216].VisStatus
    Rectangle (376,379 80x18), "ADD 20A", colour toggle: ASI02.Asi_DeviceA[20]
    Rectangle (460,397 40x20), "P217", colour variable: DataPsgForVis[217].VisStatus
    Rectangle (500,397 40x20), "P218", colour variable: DataPsgForVis[218].VisStatus
    Rectangle (460,379 80x18), "ADD 21A", colour toggle: ASI02.Asi_DeviceA[21]
    Rectangle (544,397 40x20), "P219", colour variable: DataPsgForVis[219].VisStatus
    Rectangle (584,397 40x20), "P220", colour variable: DataPsgForVis[220].VisStatus
    Rectangle (544,379 80x18), "ADD 22A", colour toggle: ASI02.Asi_DeviceA[22]
    Rectangle (628,397 40x20), "P221", colour variable: DataPsgForVis[221].VisStatus
    Rectangle (668,397 40x20), "P222", colour variable: DataPsgForVis[222].VisStatus
    Rectangle (628,379 80x18), "ADD 23A", colour toggle: ASI02.Asi_DeviceA[23]
    Rectangle (712,397 40x20), "P223", colour variable: DataPsgForVis[223].VisStatus
    Rectangle (752,397 40x20), "P224", colour variable: DataPsgForVis[224].VisStatus
    Rectangle (712,379 80x18), "ADD 24A", colour toggle: ASI02.Asi_DeviceA[24]
    Rectangle (124,440 40x20), "P225", colour variable: DataPsgForVis[225].VisStatus
    Rectangle (164,440 40x20), "P226", colour variable: DataPsgForVis[226].VisStatus
    Rectangle (124,422 80x18), "ADD 25A", colour toggle: ASI02.Asi_DeviceA[25]
    Rectangle (208,440 40x20), "P227", colour variable: DataPsgForVis[227].VisStatus
    Rectangle (248,440 40x20), "P228", colour variable: DataPsgForVis[228].VisStatus
    Rectangle (208,422 80x18), "ADD 26A", colour toggle: ASI02.Asi_DeviceA[26]
    Rectangle (292,440 40x20), "P229", colour variable: DataPsgForVis[229].VisStatus
    Rectangle (332,440 40x20), "P230", colour variable: DataPsgForVis[230].VisStatus
    Rectangle (292,422 80x18), "ADD 27A", colour toggle: ASI02.Asi_DeviceA[27]
    Rectangle (376,440 40x20), "P231", colour variable: DataPsgForVis[231].VisStatus
    Rectangle (416,440 40x20), "P232", colour variable: DataPsgForVis[232].VisStatus
    Rectangle (376,422 80x18), "ADD 28A", colour toggle: ASI02.Asi_DeviceA[28]
    Rectangle (460,440 40x20), "P233", colour variable: DataPsgForVis[233].VisStatus
    Rectangle (500,440 40x20), "P234", colour variable: DataPsgForVis[234].VisStatus
    Rectangle (460,422 80x18), "ADD 29A", colour toggle: ASI02.Asi_DeviceA[29]
    Rectangle (544,440 40x20), "P235", colour variable: DataPsgForVis[235].VisStatus
    Rectangle (584,440 40x20), "P236", colour variable: DataPsgForVis[236].VisStatus
    Rectangle (544,422 80x18), "ADD 30A", colour toggle: ASI02.Asi_DeviceA[30]
    Rectangle (628,440 40x20), "P237", colour variable: DataPsgForVis[237].VisStatus
    Rectangle (668,440 40x20), "P238", colour variable: DataPsgForVis[238].VisStatus
    Rectangle (628,422 80x18), "ADD 31A", colour toggle: ASI02.Asi_DeviceA[31]
    Rectangle (124,485 40x20), "P239", colour variable: DataPsgForVis[239].VisStatus
    Rectangle (164,485 40x20), "P240", colour variable: DataPsgForVis[240].VisStatus
    Rectangle (124,467 80x18), "ADD 01B", colour toggle: ASI02.Asi_DeviceB[1]
    Rectangle (109,524 451x21), "Timer lux"
    Rectangle (127,566 50x20), "Lux105", colour variable: DataLuxForVis[105].VisStatus
    Rectangle (177,566 40x20), "%d", text variable: DataLuxForVis[105].VisTimer, colour toggle: CronEd.CN_Sel<>CronEd.CN_Act
    Rectangle (127,606 50x20), "Lux107", colour variable: DataLuxForVis[107].VisStatus
    Rectangle (177,606 40x20), "%d", text variable: DataLuxForVis[107].VisTimer, colour toggle: CronEd.CN_Sel<>CronEd.CN_Act
    Rectangle (127,586 50x20), "Lux106", colour variable: DataLuxForVis[106].VisStatus
    Rectangle (177,586 40x20), "%d", text variable: DataLuxForVis[106].VisTimer, colour toggle: CronEd.CN_Sel<>CronEd.CN_Act
    Rectangle (127,626 50x20), "Lux108", colour variable: DataLuxForVis[108].VisStatus
    Rectangle (177,626 40x20), "%d", text variable: DataLuxForVis[108].VisTimer, colour toggle: CronEd.CN_Sel<>CronEd.CN_Act
    Rectangle (127,650 50x20), "Lux109", colour variable: DataLuxForVis[109].VisStatus
    Rectangle (177,650 40x20), "%d", text variable: DataLuxForVis[109].VisTimer, colour toggle: CronEd.CN_Sel<>CronEd.CN_Act
    Rectangle (127,670 50x20), "Lux110", colour variable: DataLuxForVis[110].VisStatus
    Rectangle (177,670 40x20), "%d", text variable: DataLuxForVis[110].VisTimer, colour toggle: CronEd.CN_Sel<>CronEd.CN_Act
    Rectangle (108,566 19x80), "13 B", colour toggle: ASI02.Asi_DeviceB[13]
    Rectangle (127,690 50x20), "Lux111", colour variable: DataLuxForVis[111].VisStatus
    Rectangle (177,690 40x20), "%d", text variable: DataLuxForVis[111].VisTimer, colour toggle: CronEd.CN_Sel<>CronEd.CN_Act
    Rectangle (127,710 50x20), "Lux112", colour variable: DataLuxForVis[112].VisStatus
    Rectangle (177,710 40x20), "%d", text variable: DataLuxForVis[112].VisTimer, colour toggle: CronEd.CN_Sel<>CronEd.CN_Act
    Rectangle (108,650 19x80), "14 B", colour toggle: ASI02.Asi_DeviceB[14]
    Rectangle (127,734 50x20), "Lux113", colour variable: DataLuxForVis[113].VisStatus
    Rectangle (177,734 40x20), "%d", text variable: DataLuxForVis[113].VisTimer, colour toggle: CronEd.CN_Sel<>CronEd.CN_Act
    Rectangle (127,754 50x20), "Lux114", colour variable: DataLuxForVis[114].VisStatus
    Rectangle (177,754 40x20), "%d", text variable: DataLuxForVis[114].VisTimer, colour toggle: CronEd.CN_Sel<>CronEd.CN_Act
    Rectangle (127,774 50x20), "Lux115", colour variable: DataLuxForVis[115].VisStatus
    Rectangle (177,774 40x20), "%d", text variable: DataLuxForVis[115].VisTimer, colour toggle: CronEd.CN_Sel<>CronEd.CN_Act
    Rectangle (127,794 50x20), "Lux116", colour variable: DataLuxForVis[116].VisStatus
    Rectangle (177,794 40x20), "%d", text variable: DataLuxForVis[116].VisTimer, colour toggle: CronEd.CN_Sel<>CronEd.CN_Act
    Rectangle (108,734 19x80), "15 B", colour toggle: ASI02.Asi_DeviceB[15]
    Rectangle (127,818 50x20), "Lux117", colour variable: DataLuxForVis[117].VisStatus
    Rectangle (177,818 40x20), "%d", text variable: DataLuxForVis[117].VisTimer, colour toggle: CronEd.CN_Sel<>CronEd.CN_Act
    Rectangle (127,838 50x20), "Lux118", colour variable: DataLuxForVis[118].VisStatus
    Rectangle (177,838 40x20), "%d", text variable: DataLuxForVis[118].VisTimer, colour toggle: CronEd.CN_Sel<>CronEd.CN_Act
    Rectangle (127,858 50x20), "Lux119", colour variable: DataLuxForVis[119].VisStatus
    Rectangle (177,858 40x20), "%d", text variable: DataLuxForVis[119].VisTimer, colour toggle: CronEd.CN_Sel<>CronEd.CN_Act
    Rectangle (127,878 50x20), "Lux120", colour variable: DataLuxForVis[120].VisStatus
    Rectangle (177,878 40x20), "%d", text variable: DataLuxForVis[120].VisTimer, colour toggle: CronEd.CN_Sel<>CronEd.CN_Act
    Rectangle (108,818 19x80), "16 B", colour toggle: ASI02.Asi_DeviceB[16]
    Rectangle (241,566 50x20), "Lux121", colour variable: DataLuxForVis[121].VisStatus
    Rectangle (291,566 40x20), "%d", text variable: DataLuxForVis[121].VisTimer, colour toggle: CronEd.CN_Sel<>CronEd.CN_Act
    Rectangle (241,586 50x20), "Lux122", colour variable: DataLuxForVis[122].VisStatus
    Rectangle (291,586 40x20), "%d", text variable: DataLuxForVis[122].VisTimer, colour toggle: CronEd.CN_Sel<>CronEd.CN_Act
    Rectangle (241,606 50x20), "Lux123", colour variable: DataLuxForVis[123].VisStatus
    Rectangle (291,606 40x20), "%d", text variable: DataLuxForVis[123].VisTimer, colour toggle: CronEd.CN_Sel<>CronEd.CN_Act
    Rectangle (241,626 50x20), "Lux124", colour variable: DataLuxForVis[124].VisStatus
    Rectangle (291,626 40x20), "%d", text variable: DataLuxForVis[124].VisTimer, colour toggle: CronEd.CN_Sel<>CronEd.CN_Act
    Rectangle (222,566 19x80), "17 B", colour toggle: ASI02.Asi_DeviceB[17]
    Rectangle (355,566 50x20), "Lux137", colour variable: DataLuxForVis[137].VisStatus
    Rectangle (405,566 40x20), "%d", text variable: DataLuxForVis[137].VisTimer, colour toggle: CronEd.CN_Sel<>CronEd.CN_Act
    Rectangle (355,586 50x20), "Lux138", colour variable: DataLuxForVis[138].VisStatus
    Rectangle (405,586 40x20), "%d", text variable: DataLuxForVis[138].VisTimer, colour toggle: CronEd.CN_Sel<>CronEd.CN_Act
    Rectangle (355,606 50x20), "Lux139", colour variable: DataLuxForVis[139].VisStatus
    Rectangle (405,606 40x20), "%d", text variable: DataLuxForVis[139].VisTimer, colour toggle: CronEd.CN_Sel<>CronEd.CN_Act
    Rectangle (355,626 50x20), "Lux140", colour variable: DataLuxForVis[140].VisStatus
    Rectangle (405,626 40x20), "%d", text variable: DataLuxForVis[140].VisTimer, colour toggle: CronEd.CN_Sel<>CronEd.CN_Act
    Rectangle (336,566 19x80), "21 B", colour toggle: ASI02.Asi_DeviceB[21]
    Rectangle (470,566 50x20), "Lux153", colour variable: DataLuxForVis[153].VisStatus
    Rectangle (520,566 40x20), "%d", text variable: DataLuxForVis[153].VisTimer, colour toggle: CronEd.CN_Sel<>CronEd.CN_Act
    Rectangle (470,586 50x20), "Lux154", colour variable: DataLuxForVis[154].VisStatus
    Rectangle (520,586 40x20), "%d", text variable: DataLuxForVis[154].VisTimer, colour toggle: CronEd.CN_Sel<>CronEd.CN_Act
    Rectangle (470,606 50x20), "Lux155", colour variable: DataLuxForVis[155].VisStatus
    Rectangle (520,606 40x20), "%d", text variable: DataLuxForVis[155].VisTimer, colour toggle: CronEd.CN_Sel<>CronEd.CN_Act
    Rectangle (470,626 50x20), "Lux156", colour variable: DataLuxForVis[156].VisStatus
    Rectangle (520,626 40x20), "%d", text variable: DataLuxForVis[156].VisTimer, colour toggle: CronEd.CN_Sel<>CronEd.CN_Act
    Rectangle (451,566 19x80), "25 B", colour toggle: ASI02.Asi_DeviceB[25]
    Rectangle (241,650 50x20), "Lux125", colour variable: DataLuxForVis[125].VisStatus
    Rectangle (291,650 40x20), "%d", text variable: DataLuxForVis[125].VisTimer, colour toggle: CronEd.CN_Sel<>CronEd.CN_Act
    Rectangle (241,670 50x20), "Lux126", colour variable: DataLuxForVis[126].VisStatus
    Rectangle (291,670 40x20), "%d", text variable: DataLuxForVis[126].VisTimer, colour toggle: CronEd.CN_Sel<>CronEd.CN_Act
    Rectangle (241,690 50x20), "Lux127", colour variable: DataLuxForVis[127].VisStatus
    Rectangle (291,690 40x20), "%d", text variable: DataLuxForVis[127].VisTimer, colour toggle: CronEd.CN_Sel<>CronEd.CN_Act
    Rectangle (241,710 50x20), "Lux128", colour variable: DataLuxForVis[128].VisStatus
    Rectangle (291,710 40x20), "%d", text variable: DataLuxForVis[124].VisTimer, colour toggle: CronEd.CN_Sel<>CronEd.CN_Act, colour variable: DataLuxForVis[128].VisStatus
    Rectangle (222,650 19x80), "18 B", colour toggle: ASI02.Asi_DeviceB[18]
    Rectangle (241,734 50x20), "Lux129", colour variable: DataLuxForVis[129].VisStatus
    Rectangle (291,734 40x20), "%d", text variable: DataLuxForVis[129].VisTimer, colour toggle: CronEd.CN_Sel<>CronEd.CN_Act
    Rectangle (241,754 50x20), "Lux130", colour variable: DataLuxForVis[130].VisStatus
    Rectangle (291,754 40x20), "%d", text variable: DataLuxForVis[130].VisTimer, colour toggle: CronEd.CN_Sel<>CronEd.CN_Act
    Rectangle (241,774 50x20), "Lux131", colour variable: DataLuxForVis[131].VisStatus
    Rectangle (291,774 40x20), "%d", text variable: DataLuxForVis[131].VisTimer, colour toggle: CronEd.CN_Sel<>CronEd.CN_Act
    Rectangle (241,794 50x20), "Lux132", colour variable: DataLuxForVis[132].VisStatus
    Rectangle (291,794 40x20), "%d", text variable: DataLuxForVis[132].VisTimer, colour toggle: CronEd.CN_Sel<>CronEd.CN_Act
    Rectangle (222,734 19x80), "19 B", colour toggle: ASI02.Asi_DeviceB[19]
    Rectangle (241,818 50x20), "Lux133", colour variable: DataLuxForVis[133].VisStatus
    Rectangle (291,818 40x20), "%d", text variable: DataLuxForVis[133].VisTimer, colour toggle: CronEd.CN_Sel<>CronEd.CN_Act
    Rectangle (241,838 50x20), "Lux134", colour variable: DataLuxForVis[134].VisStatus
    Rectangle (291,838 40x20), "%d", text variable: DataLuxForVis[134].VisTimer, colour toggle: CronEd.CN_Sel<>CronEd.CN_Act
    Rectangle (241,858 50x20), "Lux135", colour variable: DataLuxForVis[135].VisStatus
    Rectangle (291,858 40x20), "%d", text variable: DataLuxForVis[135].VisTimer, colour toggle: CronEd.CN_Sel<>CronEd.CN_Act
    Rectangle (241,878 50x20), "Lux136", colour variable: DataLuxForVis[136].VisStatus
    Rectangle (291,878 40x20), "%d", text variable: DataLuxForVis[136].VisTimer, colour toggle: CronEd.CN_Sel<>CronEd.CN_Act
    Rectangle (222,818 19x80), "20 B", colour toggle: ASI02.Asi_DeviceB[20]
    Rectangle (355,650 50x20), "Lux141", colour variable: DataLuxForVis[141].VisStatus
    Rectangle (405,650 40x20), "%d", text variable: DataLuxForVis[141].VisTimer, colour toggle: CronEd.CN_Sel<>CronEd.CN_Act
    Rectangle (355,670 50x20), "Lux142", colour variable: DataLuxForVis[142].VisStatus
    Rectangle (405,670 40x20), "%d", text variable: DataLuxForVis[142].VisTimer, colour toggle: CronEd.CN_Sel<>CronEd.CN_Act
    Rectangle (355,690 50x20), "Lux143", colour variable: DataLuxForVis[143].VisStatus
    Rectangle (405,690 40x20), "%d", text variable: DataLuxForVis[143].VisTimer, colour toggle: CronEd.CN_Sel<>CronEd.CN_Act
    Rectangle (355,710 50x20), "Lux144", colour variable: DataLuxForVis[144].VisStatus
    Rectangle (405,710 40x20), "%d", text variable: DataLuxForVis[144].VisTimer, colour toggle: CronEd.CN_Sel<>CronEd.CN_Act
    Rectangle (336,650 19x80), "22 B", colour toggle: ASI02.Asi_DeviceB[22]
    Rectangle (355,734 50x20), "Lux145", colour variable: DataLuxForVis[145].VisStatus
    Rectangle (405,734 40x20), "%d", text variable: DataLuxForVis[145].VisTimer, colour toggle: CronEd.CN_Sel<>CronEd.CN_Act
    Rectangle (355,754 50x20), "Lux146", colour variable: DataLuxForVis[146].VisStatus
    Rectangle (405,754 40x20), "%d", text variable: DataLuxForVis[146].VisTimer, colour toggle: CronEd.CN_Sel<>CronEd.CN_Act
    Rectangle (355,774 50x20), "Lux147", colour variable: DataLuxForVis[147].VisStatus
    Rectangle (405,774 40x20), "%d", text variable: DataLuxForVis[147].VisTimer, colour toggle: CronEd.CN_Sel<>CronEd.CN_Act
    Rectangle (355,794 50x20), "Lux148", colour variable: DataLuxForVis[148].VisStatus
    Rectangle (405,794 40x20), "%d", text variable: DataLuxForVis[148].VisTimer, colour toggle: CronEd.CN_Sel<>CronEd.CN_Act
    Rectangle (336,734 19x80), "23 B", colour toggle: ASI02.Asi_DeviceB[23]
    Rectangle (355,818 50x20), "Lux149", colour variable: DataLuxForVis[149].VisStatus
    Rectangle (405,818 40x20), "%d", text variable: DataLuxForVis[149].VisTimer, colour toggle: CronEd.CN_Sel<>CronEd.CN_Act
    Rectangle (355,838 50x20), "Lux150", colour variable: DataLuxForVis[150].VisStatus
    Rectangle (405,838 40x20), "%d", text variable: DataLuxForVis[150].VisTimer, colour toggle: CronEd.CN_Sel<>CronEd.CN_Act
    Rectangle (355,858 50x20), "Lux151", colour variable: DataLuxForVis[151].VisStatus
    Rectangle (405,858 40x20), "%d", text variable: DataLuxForVis[151].VisTimer, colour toggle: CronEd.CN_Sel<>CronEd.CN_Act
    Rectangle (355,878 50x20), "Lux152", colour variable: DataLuxForVis[152].VisStatus
    Rectangle (405,878 40x20), "%d", text variable: DataLuxForVis[152].VisTimer, colour toggle: CronEd.CN_Sel<>CronEd.CN_Act
        OnMouseDown: write the text variable via Edit, min 10, max 32760, title '1'
    Rectangle (336,818 19x80), "24 B", colour toggle: ASI02.Asi_DeviceB[24]
    Rectangle (470,650 50x20), "Lux157", colour variable: DataLuxForVis[157].VisStatus
    Rectangle (520,650 40x20), "%d", text variable: DataLuxForVis[157].VisTimer, colour toggle: CronEd.CN_Sel<>CronEd.CN_Act
    Rectangle (470,670 50x20), "Lux158", colour variable: DataLuxForVis[158].VisStatus
    Rectangle (520,670 40x20), "%d", text variable: DataLuxForVis[158].VisTimer, colour toggle: CronEd.CN_Sel<>CronEd.CN_Act
    Rectangle (470,690 50x20), "Lux159", colour variable: DataLuxForVis[159].VisStatus
    Rectangle (520,690 40x20), "%d", text variable: DataLuxForVis[159].VisTimer, colour toggle: CronEd.CN_Sel<>CronEd.CN_Act
    Rectangle (470,710 50x20), "Lux160", colour variable: DataLuxForVis[160].VisStatus
    Rectangle (520,710 40x20), "%d", text variable: DataLuxForVis[160].VisTimer, colour toggle: CronEd.CN_Sel<>CronEd.CN_Act
    Rectangle (451,650 19x80), "26 B", colour toggle: ASI02.Asi_DeviceB[26]
    Group (470,734 90x20)
        Rectangle (0,0 50x20), "Lux161", colour variable: DataLuxForVis[161].VisStatus
        Rectangle (50,0 40x20), "%d", text variable: DataLuxForVis[161].VisTimer, colour toggle: CronEd.CN_Sel<>CronEd.CN_Act
    Group (470,754 90x20)
        Rectangle (0,0 50x20), "Lux162", colour variable: DataLuxForVis[162].VisStatus
        Rectangle (50,0 40x20), "%d", text variable: DataLuxForVis[162].VisTimer, colour toggle: CronEd.CN_Sel<>CronEd.CN_Act
    Group (470,774 90x20)
        Rectangle (0,0 50x20), "Lux163", colour variable: DataLuxForVis[163].VisStatus
        Rectangle (50,0 40x20), "%d", text variable: DataLuxForVis[163].VisTimer, colour toggle: CronEd.CN_Sel<>CronEd.CN_Act
    Group (470,794 90x20)
        Rectangle (0,0 50x20), "Lux164", colour variable: DataLuxForVis[164].VisStatus
        Rectangle (50,0 40x20), "%d", text variable: DataLuxForVis[164].VisTimer, colour toggle: CronEd.CN_Sel<>CronEd.CN_Act
    Rectangle (451,734 19x80), "27 B", colour toggle: ASI02.Asi_DeviceB[27]
    Group (470,818 90x20)
        Rectangle (0,0 50x20), "Lux165", colour variable: DataLuxForVis[165].VisStatus
        Rectangle (50,0 40x20), "%d", text variable: DataLuxForVis[165].VisTimer, colour toggle: CronEd.CN_Sel<>CronEd.CN_Act
    Group (470,838 90x20)
        Rectangle (0,0 50x20), "Lux166", colour variable: DataLuxForVis[166].VisStatus
        Rectangle (50,0 40x20), "%d", text variable: DataLuxForVis[166].VisTimer, colour toggle: CronEd.CN_Sel<>CronEd.CN_Act
    Group (470,858 90x20)
        Rectangle (0,0 50x20), "Lux167", colour variable: DataLuxForVis[167].VisStatus
        Rectangle (50,0 40x20), "%d", text variable: DataLuxForVis[167].VisTimer, colour toggle: CronEd.CN_Sel<>CronEd.CN_Act
    Group (470,878 90x20)
        Rectangle (0,0 50x20), "Lux168", colour variable: DataLuxForVis[168].VisStatus
        Rectangle (50,0 40x20), "%d", text variable: DataLuxForVis[168].VisTimer, colour toggle: CronEd.CN_Sel<>CronEd.CN_Act
    Rectangle (451,818 19x80), "28 B", colour toggle: ASI02.Asi_DeviceB[28]
    Rectangle (109,547 451x17), "ASI 2"
    Rectangle (108,936 115x17), "ASI 1"
    Rectangle (108,912 467x21), "Crono lux"
    Rectangle (133,955 50x20), "Lux046", colour variable: DataLuxForVis[46].VisStatus
    Rectangle (183,955 40x20), "%d", text variable: DataLuxForVis[46].VisMod, colour toggle: CronEd.CN_Sel<>CronEd.CN_Act
    Rectangle (133,975 50x20), "Lux047", colour variable: DataLuxForVis[47].VisStatus
    Rectangle (183,975 40x20), "%d", text variable: DataLuxForVis[47].VisMod, colour toggle: CronEd.CN_Sel<>CronEd.CN_Act
    Rectangle (133,995 50x20), "Lux048", colour variable: DataLuxForVis[48].VisStatus
    Rectangle (183,995 40x20), "%d", text variable: DataLuxForVis[48].VisMod, colour toggle: CronEd.CN_Sel<>CronEd.CN_Act
    Rectangle (108,955 25x20), "02B", colour toggle: ASI01.Asi_DeviceB[2]
    Rectangle (108,975 25x20), "03B", colour toggle: ASI01.Asi_DeviceB[3]
    Rectangle (108,995 25x20), "04B", colour toggle: ASI01.Asi_DeviceB[4]
    Rectangle (226,936 349x17), "ASI 2"
    Rectangle (251,955 50x20), "Lux07", colour variable: DataLuxForVis[7].VisStatus
    Rectangle (301,955 40x20), "%d", text variable: DataLuxForVis[7].VisMod, colour toggle: CronEd.CN_Sel<>CronEd.CN_Act
    Rectangle (226,955 25x20), "02B", colour toggle: ASI02.Asi_DeviceB[2]
    Rectangle (226,975 25x20), "02B", colour toggle: ASI02.Asi_DeviceB[2]
    Rectangle (251,975 50x20), "Lux08", colour variable: DataLuxForVis[8].VisStatus
    Rectangle (301,975 40x20), "%d", text variable: DataLuxForVis[8].VisMod, colour toggle: CronEd.CN_Sel<>CronEd.CN_Act
    Rectangle (226,995 25x20), "03B", colour toggle: ASI02.Asi_DeviceB[3]
    Rectangle (251,995 50x20), "Lux09", colour variable: DataLuxForVis[9].VisStatus
    Rectangle (301,995 40x20), "%d", text variable: DataLuxForVis[9].VisMod, colour toggle: CronEd.CN_Sel<>CronEd.CN_Act
    Rectangle (226,1015 25x20), "03B", colour toggle: ASI02.Asi_DeviceB[3]
    Rectangle (251,1015 50x20), "Lux10", colour variable: DataLuxForVis[10].VisStatus
    Rectangle (301,1015 40x20), "%d", text variable: DataLuxForVis[10].VisMod, colour toggle: CronEd.CN_Sel<>CronEd.CN_Act
    Rectangle (251,1035 50x20), "Lux11", colour variable: DataLuxForVis[11].VisStatus
    Rectangle (301,1035 40x20), "%d", text variable: DataLuxForVis[11].VisMod, colour toggle: CronEd.CN_Sel<>CronEd.CN_Act
    Rectangle (226,1035 25x20), "04B", colour toggle: ASI02.Asi_DeviceB[4]
    Rectangle (226,1055 25x20), "04B", colour toggle: ASI02.Asi_DeviceB[4]
    Rectangle (251,1055 50x20), "Lux12", colour variable: DataLuxForVis[12].VisStatus
    Rectangle (301,1055 40x20), "%d", text variable: DataLuxForVis[12].VisMod, colour toggle: CronEd.CN_Sel<>CronEd.CN_Act
    Rectangle (226,1075 25x20), "05B", colour toggle: ASI02.Asi_DeviceB[5]
    Rectangle (251,1075 50x20), "Lux27", colour variable: DataLuxForVis[27].VisStatus
    Rectangle (301,1075 40x20), "%d", text variable: DataLuxForVis[27].VisMod, colour toggle: CronEd.CN_Sel<>CronEd.CN_Act
    Rectangle (226,1095 25x20), "05B", colour toggle: ASI02.Asi_DeviceB[5]
    Rectangle (251,1095 50x20), "Lux28", colour variable: DataLuxForVis[28].VisStatus
    Rectangle (301,1095 40x20), "%d", text variable: DataLuxForVis[28].VisMod, colour toggle: CronEd.CN_Sel<>CronEd.CN_Act
    Rectangle (251,1115 50x20), "Lux29", colour variable: DataLuxForVis[29].VisStatus
    Rectangle (301,1115 40x20), "%d", text variable: DataLuxForVis[29].VisMod, colour toggle: CronEd.CN_Sel<>CronEd.CN_Act
    Rectangle (226,1115 25x20), "06B", colour toggle: ASI02.Asi_DeviceB[6]
    Rectangle (226,1135 25x20), "06B", colour toggle: ASI02.Asi_DeviceB[6]
    Rectangle (251,1135 50x20), "Lux30", colour variable: DataLuxForVis[30].VisStatus
    Rectangle (301,1135 40x20), "%d", text variable: DataLuxForVis[30].VisMod, colour toggle: CronEd.CN_Sel<>CronEd.CN_Act
    Rectangle (344,955 25x20), "07B", colour toggle: ASI02.Asi_DeviceB[7]
    Rectangle (369,955 50x20), "Lux31", colour variable: DataLuxForVis[31].VisStatus
    Rectangle (419,955 40x20), "%d", text variable: DataLuxForVis[31].VisMod, colour toggle: CronEd.CN_Sel<>CronEd.CN_Act
    Rectangle (344,975 25x20), "07B", colour toggle: ASI02.Asi_DeviceB[7]
    Rectangle (369,975 50x20), "Lux32", colour variable: DataLuxForVis[32].VisStatus
    Rectangle (419,975 40x20), "%d", text variable: DataLuxForVis[32].VisMod, colour toggle: CronEd.CN_Sel<>CronEd.CN_Act
    Rectangle (369,995 50x20), "Lux33", colour variable: DataLuxForVis[33].VisStatus
    Rectangle (419,995 40x20), "%d", text variable: DataLuxForVis[33].VisMod, colour toggle: CronEd.CN_Sel<>CronEd.CN_Act
    Rectangle (344,995 25x20), "08B", colour toggle: ASI02.Asi_DeviceB[8]
    Rectangle (344,1015 25x20), "08B", colour toggle: ASI02.Asi_DeviceB[8]
    Rectangle (369,1015 50x20), "Lux34", colour variable: DataLuxForVis[34].VisStatus
    Rectangle (419,1015 40x20), "%d", text variable: DataLuxForVis[34].VisMod, colour toggle: CronEd.CN_Sel<>CronEd.CN_Act
    Rectangle (344,1035 25x20), "09B", colour toggle: ASI02.Asi_DeviceB[9]
    Rectangle (369,1035 50x20), "Lux35", colour variable: DataLuxForVis[35].VisStatus
    Rectangle (419,1035 40x20), "%d", text variable: DataLuxForVis[35].VisMod, colour toggle: CronEd.CN_Sel<>CronEd.CN_Act
    Rectangle (344,1055 25x20), "09B", colour toggle: ASI02.Asi_DeviceB[9]
    Rectangle (369,1055 50x20), "Lux36", colour variable: DataLuxForVis[36].VisStatus
    Rectangle (419,1055 40x20), "%d", text variable: DataLuxForVis[36].VisMod, colour toggle: CronEd.CN_Sel<>CronEd.CN_Act
    Rectangle (369,1075 50x20), "Lux37", colour variable: DataLuxForVis[37].VisStatus
    Rectangle (419,1075 40x20), "%d", text variable: DataLuxForVis[37].VisMod, colour toggle: CronEd.CN_Sel<>CronEd.CN_Act
    Rectangle (344,1075 25x20), "10B", colour toggle: ASI02.Asi_DeviceB[10]
    Rectangle (344,1095 25x20), "10B", colour toggle: ASI02.Asi_DeviceB[10]
    Rectangle (369,1095 50x20), "Lux38", colour variable: DataLuxForVis[38].VisStatus
    Rectangle (419,1095 40x20), "%d", text variable: DataLuxForVis[38].VisMod, colour toggle: CronEd.CN_Sel<>CronEd.CN_Act
    Rectangle (344,1115 25x20), "11B", colour toggle: ASI02.Asi_DeviceB[11]
    Rectangle (369,1115 50x20), "Lux39", colour variable: DataLuxForVis[39].VisStatus
    Rectangle (419,1115 40x20), "%d", text variable: DataLuxForVis[39].VisMod, colour toggle: CronEd.CN_Sel<>CronEd.CN_Act
    Rectangle (344,1135 25x20), "11B", colour toggle: ASI02.Asi_DeviceB[11]
    Rectangle (369,1135 50x20), "Lux40", colour variable: DataLuxForVis[40].VisStatus
    Rectangle (419,1135 40x20), "%d", text variable: DataLuxForVis[40].VisMod, colour toggle: CronEd.CN_Sel<>CronEd.CN_Act
    Rectangle (486,955 50x20), "Lux41", colour variable: DataLuxForVis[41].VisStatus
    Rectangle (536,955 40x20), "%d", text variable: DataLuxForVis[41].VisMod, colour toggle: CronEd.CN_Sel<>CronEd.CN_Act
    Rectangle (461,955 25x20), "12B", colour toggle: ASI02.Asi_DeviceA[12]
    Rectangle (461,975 25x20), "12B", colour toggle: ASI02.Asi_DeviceA[12]
    Rectangle (486,975 50x20), "Lux42", colour variable: DataLuxForVis[42].VisStatus
    Rectangle (536,975 40x20), "%d", text variable: DataLuxForVis[42].VisMod, colour toggle: CronEd.CN_Sel<>CronEd.CN_Act
    Rectangle (124,74 40x20), "P089", invisible if: FALSE, colour variable: DataPsgForVis[89].VisStatus
    Rectangle (164,74 40x20), "P090", colour variable: DataPsgForVis[90].VisStatus
    Rectangle (124,56 80x18), "ADD 01A", colour toggle: ASI01.Asi_DeviceA[1]
    Rectangle (208,74 40x20), "P091", colour variable: DataPsgForVis[91].VisStatus
    Rectangle (248,74 40x20), "P092", colour variable: DataPsgForVis[92].VisStatus
    Rectangle (208,56 80x18), "ADD 02A", colour toggle: ASI01.Asi_DeviceA[2]
    Rectangle (292,74 40x20), "P093", colour variable: DataPsgForVis[93].VisStatus
    Rectangle (332,74 40x20), "P094", colour variable: DataPsgForVis[94].VisStatus
    Rectangle (292,56 80x18), "ADD 03A", colour toggle: ASI01.Asi_DeviceA[3]
    Rectangle (376,74 40x20), "P095", colour variable: DataPsgForVis[95].VisStatus
    Rectangle (416,74 40x20), "P096", colour variable: DataPsgForVis[96].VisStatus
    Rectangle (376,56 80x18), "ADD 04A", colour toggle: ASI01.Asi_DeviceA[4]
    Rectangle (460,74 40x20), "P097", colour variable: DataPsgForVis[97].VisStatus
    Rectangle (500,74 40x20), "P098", colour variable: DataPsgForVis[98].VisStatus
    Rectangle (460,56 80x18), "ADD 05A", colour toggle: ASI01.Asi_DeviceA[5]
    Rectangle (544,74 40x20), "P099", colour variable: DataPsgForVis[99].VisStatus
    Rectangle (584,74 40x20), "P100", colour variable: DataPsgForVis[100].VisStatus
    Rectangle (544,56 80x18), "ADD 06A", colour toggle: ASI01.Asi_DeviceA[6]
    Rectangle (628,74 40x20), "P101", colour variable: DataPsgForVis[101].VisStatus
    Rectangle (668,74 40x20), "P102", colour variable: DataPsgForVis[102].VisStatus
    Rectangle (628,56 80x18), "ADD 07A", colour toggle: ASI01.Asi_DeviceA[7]
    Rectangle (712,74 40x20), "P103", colour variable: DataPsgForVis[103].VisStatus
    Rectangle (752,74 40x20), "P104", colour variable: DataPsgForVis[104].VisStatus
    Rectangle (712,56 80x18), "ADD 08A", colour toggle: ASI01.Asi_DeviceA[8]
    Rectangle (712,117 40x20), "P119", colour variable: DataPsgForVis[119].VisStatus
    Rectangle (752,117 40x20), "P120", colour variable: DataPsgForVis[120].VisStatus
    Rectangle (712,99 80x18), "ADD 16A", colour toggle: ASI01.Asi_DeviceA[16]
    Rectangle (124,117 40x20), "P105", colour variable: DataPsgForVis[105].VisStatus
    Rectangle (164,117 40x20), "P106", colour variable: DataPsgForVis[106].VisStatus
    Rectangle (124,99 80x18), "ADD 09A", colour toggle: ASI01.Asi_DeviceA[9]
    Rectangle (208,117 40x20), "P107", colour variable: DataPsgForVis[107].VisStatus
    Rectangle (248,117 40x20), "P108", colour variable: DataPsgForVis[108].VisStatus
    Rectangle (208,99 80x18), "ADD 10A", colour toggle: ASI01.Asi_DeviceA[10]
    Rectangle (292,117 40x20), "P109", colour variable: DataPsgForVis[109].VisStatus
    Rectangle (332,117 40x20), "P110", colour variable: DataPsgForVis[110].VisStatus
    Rectangle (292,99 80x18), "ADD 11A", colour toggle: ASI01.Asi_DeviceA[11]
    Rectangle (376,117 40x20), "P111", colour variable: DataPsgForVis[111].VisStatus
    Rectangle (416,117 40x20), "P112", colour variable: DataPsgForVis[112].VisStatus
    Rectangle (376,99 80x18), "ADD 12A", colour toggle: ASI01.Asi_DeviceA[12]
    Rectangle (460,117 40x20), "P113", colour variable: DataPsgForVis[113].VisStatus
    Rectangle (500,117 40x20), "P114", colour variable: DataPsgForVis[114].VisStatus
    Rectangle (460,99 80x18), "ADD 13A", colour toggle: ASI01.Asi_DeviceA[13]
    Rectangle (544,117 40x20), "P115", colour variable: DataPsgForVis[115].VisStatus
    Rectangle (584,117 40x20), "P116", colour variable: DataPsgForVis[116].VisStatus
    Rectangle (544,99 80x18), "ADD 14A", colour toggle: ASI01.Asi_DeviceA[14]
    Rectangle (628,117 40x20), "P117", colour variable: DataPsgForVis[117].VisStatus
    Rectangle (668,117 40x20), "P118", colour variable: DataPsgForVis[118].VisStatus
    Rectangle (628,99 80x18), "ADD 15A", colour toggle: ASI01.Asi_DeviceA[15]
    Rectangle (712,160 40x20), "P163", colour variable: DataPsgForVis[163].VisStatus
    Rectangle (752,160 40x20), "P164", colour variable: DataPsgForVis[164].VisStatus
    Rectangle (712,142 80x18), "ADD 24A", colour toggle: ASI01.Asi_DeviceA[24]
    Rectangle (124,160 40x20), "P149", colour variable: DataPsgForVis[149].VisStatus
    Rectangle (164,160 40x20), "P150", colour variable: DataPsgForVis[150].VisStatus
    Rectangle (124,142 80x18), "ADD 17A", colour toggle: ASI01.Asi_DeviceA[17]
    Rectangle (208,160 40x20), "P151", colour variable: DataPsgForVis[151].VisStatus
    Rectangle (248,160 40x20), "P152", colour variable: DataPsgForVis[152].VisStatus
    Rectangle (208,142 80x18), "ADD 18A", colour toggle: ASI01.Asi_DeviceA[18]
    Rectangle (292,160 40x20), "P153", colour variable: DataPsgForVis[153].VisStatus
    Rectangle (332,160 40x20), "P154", colour variable: DataPsgForVis[154].VisStatus
    Rectangle (292,142 80x18), "ADD 19A", colour toggle: ASI01.Asi_DeviceA[19]
    Rectangle (376,160 40x20), "P155", colour variable: DataPsgForVis[155].VisStatus
    Rectangle (416,160 40x20), "P156", colour variable: DataPsgForVis[156].VisStatus
    Rectangle (376,142 80x18), "ADD 20A", colour toggle: ASI01.Asi_DeviceA[20]
    Rectangle (460,160 40x20), "P157", colour variable: DataPsgForVis[157].VisStatus
    Rectangle (500,160 40x20), "P158", colour variable: DataPsgForVis[158].VisStatus
    Rectangle (460,142 80x18), "ADD 21A", colour toggle: ASI01.Asi_DeviceA[21]
    Rectangle (544,160 40x20), "P159", colour variable: DataPsgForVis[159].VisStatus
    Rectangle (584,160 40x20), "P160", colour variable: DataPsgForVis[160].VisStatus
    Rectangle (544,142 80x18), "ADD 22A", colour toggle: ASI01.Asi_DeviceA[22]
    Rectangle (628,160 40x20), "P161", colour variable: DataPsgForVis[161].VisStatus
    Rectangle (668,160 40x20), "P162", colour variable: DataPsgForVis[162].VisStatus
    Rectangle (628,142 80x18), "ADD 23A", colour toggle: ASI01.Asi_DeviceA[23]
    Rectangle (124,246 40x20), "P179", colour variable: DataPsgForVis[179].VisStatus
    Rectangle (164,246 40x20), "P180", colour variable: DataPsgForVis[180].VisStatus
    Rectangle (124,228 80x18), "ADD 01B", colour toggle: ASI01.Asi_DeviceB[1]
    Rectangle (124,203 40x20), "P165", colour variable: DataPsgForVis[165].VisStatus
    Rectangle (164,203 40x20), "P166", colour variable: DataPsgForVis[166].VisStatus
    Rectangle (124,185 80x18), "ADD 25A", colour toggle: ASI01.Asi_DeviceA[25]
    Rectangle (208,203 40x20), "P167", colour variable: DataPsgForVis[167].VisStatus
    Rectangle (248,203 40x20), "P168", colour variable: DataPsgForVis[168].VisStatus
    Rectangle (208,185 80x18), "ADD 26A", colour toggle: ASI01.Asi_DeviceA[26]
    Rectangle (292,203 40x20), "P169", colour variable: DataPsgForVis[169].VisStatus
    Rectangle (332,203 40x20), "P170", colour variable: DataPsgForVis[170].VisStatus
    Rectangle (292,185 80x18), "ADD 27A", colour toggle: ASI01.Asi_DeviceA[27]
    Rectangle (376,203 40x20), "P171", colour variable: DataPsgForVis[171].VisStatus
    Rectangle (416,203 40x20), "P172", colour variable: DataPsgForVis[172].VisStatus
    Rectangle (376,185 80x18), "ADD 28A", colour toggle: ASI01.Asi_DeviceA[28]
    Rectangle (460,203 40x20), "P173", colour variable: DataPsgForVis[173].VisStatus
    Rectangle (500,203 40x20), "P174", colour variable: DataPsgForVis[174].VisStatus
    Rectangle (460,185 80x18), "ADD 29A", colour toggle: ASI01.Asi_DeviceA[29]
    Rectangle (544,203 40x20), "P175", colour variable: DataPsgForVis[175].VisStatus
    Rectangle (584,203 40x20), "P176", colour variable: DataPsgForVis[176].VisStatus
    Rectangle (544,185 80x18), "ADD 30A", colour toggle: ASI01.Asi_DeviceA[30]
    Rectangle (628,203 40x20), "P177", colour variable: DataPsgForVis[177].VisStatus
    Rectangle (668,203 40x20), "P178", colour variable: DataPsgForVis[178].VisStatus
    Rectangle (628,185 80x18), "ADD 31A", colour toggle: ASI01.Asi_DeviceA[31]
    Rectangle (568,524 156x21), "Timer lux modify"
    Rectangle (568,547 156x112)
    Rectangle (574,553 60x20), "LUX Nr."
    Rectangle (634,553 40x20), "%d", text variable: PLC_PRG.TimerLuxSelected
        OnMouseDown: write the text variable via Edit, min 1, max LUXM_MAX_ID, title '1'
    Rectangle (634,574 40x20), "%d", text variable: DataLuxForVis[PLC_PRG.TimerLuxSelected].VisTimer
    Rectangle (574,574 60x20), "Timer (s)"
    Button (574,632 137x20), "Change timer"
        OnMouseClick:  ToggleVariable=PLC_PRG.VisModify_T_Lux
    Rectangle (672,603 40x20), "%d", text variable: PLC_PRG.TimerLuxValue
        OnMouseDown: write the text variable via Edit, min 1, max 65000, title '1'
    Rectangle (574,603 97x20), "New value (s)"
    Rectangle (584,913 152x21), "On/Off Lux"
    Group (584,937 152x112)
        Rectangle (0,0 152x112)
        Rectangle (3,4 60x20), "LUX Nr."
        Rectangle (63,4 40x20), "%d", text variable: PLC_PRG.VisLuxOnOffSelected
            OnMouseDown: write the text variable via Edit, min 1, max LUXM_MAX_ID, title '1'
        Button (8,86 137x20), "Change mode"
            OnMouseClick:  ToggleVariable=PLC_PRG.VisModify_Man_Lux
        Rectangle (3,30 39x53), "Aut Man"
        DipSwitch (33,39 40x43), variable: PLC_PRG.VisValueManAut, behaviour: TOGGLE, style: Switch-DipSwitch-Gray
        Rectangle (75,30 39x53), "On Off"
        DipSwitch (104,39 40x43), variable: PLC_PRG.VisValueManOnOff, behaviour: TOGGLE, style: Switch-DipSwitch-Gray
    Rectangle (585,1056 107x95), "Mode: 00 - Man Off 01 - Man On 02 - Aut Cron 03 - Aut Timer"
    Button (731,11 60x30), "Crono"
        OnMouseUp:  Assign=VIS_CHONOEDITOR, Type=Assignment
    Rectangle (125,11 586x30), "%s === Visualization", text variable: Plant_NAME
    Rectangle (568,670 156x52), "Green - OK, Off Light Green - OK, On Red - Asi slave Error", invisible if: 0
    Rectangle (2,80 119x32), "Green - ASi OK Yellow - Asi Warning", invisible if: 0
    Rectangle (19,13 98x27), "PLC # %s", text variable: PLC_ID
END_VISUALIZATION
